//! <summary>Borrows the concrete class name for the instance lifetime. Callers must not modify it.</summary>
{attribute 'monitoring' := 'call'}
PROPERTY ClassName : REFERENCE TO STRING
GET
ClassName REF= _ClassName;
END_GET
END_PROPERTY

//! <summary>Borrows the compiler-initialized namespace. Callers must not modify it.</summary>
{attribute 'monitoring' := 'call'}
PROPERTY NamespaceName : REFERENCE TO STRING
GET
NamespaceName REF= CurrentNamespace.Name;
END_GET
END_PROPERTY

//! <summary>Reports the complete instance size in bytes, excluding separately allocated storage.</summary>
{attribute 'monitoring' := 'call'}
PROPERTY SelfSize : ULINT
GET
SelfSize := XSIZEOF(THIS^);
END_GET
END_PROPERTY

END_FUNCTION_BLOCK

// ---- Tests/Loggers/LoggerIntegrationTestGroup.TcPOU
(*
SPDX-FileCopyrightText: c 2026 Oleksandr Tiutyk <trofimich@gmail.com>
SPDX-License-Identifier: MIT
License: https://opensource.org/license/mit
*)

(*!
<summary>Groups file rotation, unfiltered file routing and native event delivery.</summary>
<description>
Owns five children in a fixed array for single-task use. Children borrows that array. The group must not be
copied.
</description>
*)

{attribute 'no_assign'}
{attribute 'no_explicit_call' := 'do not call this function block directly'}
FUNCTION_BLOCK LoggerIntegrationTestGroup EXTENDS TOF_Testing.TestGroup<5>
VAR_STAT
	{attribute 'hide'}
	_ClassName : STRING := __POUNAME();
END_VAR
VAR
	_FileRotation : TextFileLoggerRotationTest(name := "TextFileRotation", parent := THIS^);
	_EventCategories : EventLoggerCategoryTest(name := "EventCategories", parent := THIS^);
	_QueuedEvents : QueuedEventLoggerTest(name := "QueuedEvents", parent := THIS^);

	_DirectDirectory : LoggerTestDirectory(
		directoryPath := 'C:\OpenFrameworkTests\Logger_Direct',
		logFilePrefix := 'Probe'
	);
	_DirectFileLogger : TOF_Loggers.SimpleTextFileLogger(
		directoryPath := 'C:\OpenFrameworkTests\Logger_Direct',
		logFilePrefix := 'Probe',
		maxRecordsPerFile := 1,
		directoryPathType := Tc2_System.E_OpenPath.PATH_GENERIC,
		timeout := T#2S,
		amsNetId := ''
	);
	_DirectRouting : LoggerRoutingTest(
		name := "DirectFileFeedbackAndReadback",
		parent := THIS^,
		fileLogger := _DirectFileLogger,
		directory := _DirectDirectory,
		queue := 0
	);

	_QueuedDirectory : LoggerTestDirectory(
		directoryPath := 'C:\OpenFrameworkTests\Logger_Queued',
		logFilePrefix := 'Probe'
	);
	_QueuedFileLogger : TOF_Loggers.SimpleTextFileLogger(
		directoryPath := 'C:\OpenFrameworkTests\Logger_Queued',
		logFilePrefix := 'Probe',
		maxRecordsPerFile := 1,
		directoryPathType := Tc2_System.E_OpenPath.PATH_GENERIC,
		timeout := T#2S,
		amsNetId := ''
	);
	_Queue : TOF_Loggers.QueuedLogger;
	_QueuedRouting : LoggerRoutingTest(
		name := "QueuedFileFeedbackAndReadback",
		parent := THIS^,
		fileLogger := _QueuedFileLogger,
		directory := _QueuedDirectory,
		queue := _Queue
	);

	_Children : ARRAY [0.._ChildCount - 1] OF TOF_Testing.ITestElement :=
		[_FileRotation, _EventCategories, _QueuedEvents, _DirectRouting, _QueuedRouting];
END_VAR

//! <summary>Borrows the fixed child array. Callers must not modify it.</summary>
{attribute 'monitoring' := 'call'}
PROPERTY Children : REFERENCE TO ARRAY [0.._ChildCount - 1] OF TOF_Testing.ITestElement
GET
Children REF= _Children;
END_GET
END_PROPERTY

//! <summary>Borrows the concrete class name for the instance lifetime. Callers must not modify it.</summary>
{attribute 'monitoring' := 'call'}
PROPERTY ClassName : REFERENCE TO STRING
GET
ClassName REF= _ClassName;
END_GET
END_PROPERTY

//! <summary>Borrows the compiler-initialized namespace. Callers must not modify it.</summary>
{attribute 'monitoring' := 'call'}
PROPERTY NamespaceName : REFERENCE TO STRING
GET
NamespaceName REF= CurrentNamespace.Name;
END_GET
END_PROPERTY

//! <summary>Reports the complete instance size in bytes, excluding separately allocated storage.</summary>
{attribute 'monitoring' := 'call'}
PROPERTY SelfSize : ULINT
GET
SelfSize := XSIZEOF(THIS^);
END_GET
END_PROPERTY

END_FUNCTION_BLOCK

// ---- Tests/Loggers/TextFileLoggerRotationTest.TcPOU
(*
SPDX-FileCopyrightText: c 2026 Oleksandr Tiutyk <trofimich@gmail.com>
SPDX-License-Identifier: MIT
License: https://opensource.org/license/mit
*)

(*!
<summary>Checks numbered UTF-16 records and file rotation in an exclusively owned directory.</summary>
<description>
One task writes 49 records, stops the logger and reads the five generated files before removal.
A 30-second scenario deadline includes preparation and readback. Failures retain cooperative cleanup
without a forced deadline. Reset the runner only after completion.
</description>
*)

{attribute 'no_assign'}
{attribute 'no_explicit_call' := 'do not call this function block directly'}
FUNCTION_BLOCK TextFileLoggerRotationTest EXTENDS TOF_Testing.MultiCycleTest
VAR_STAT
	{attribute 'hide'}
	_ClassName : STRING := __POUNAME();
END_VAR
VAR
	_SimpleTextFileLogger : TOF_Loggers.SimpleTextFileLogger(
		directoryPath := 'C:\OpenFrameworkTests\Logger_Smoke',
		logFilePrefix := 'Log',
		maxRecordsPerFile := 10,
		directoryPathType := Tc2_System.E_OpenPath.PATH_GENERIC,
		timeout := Tc2_System.Global_Variables.DEFAULT_ADS_TIMEOUT,
		amsNetId := ''
	);
	_LogDirectory : LoggerTestDirectory(
		directoryPath := 'C:\OpenFrameworkTests\Logger_Smoke',
		logFilePrefix := 'Log'
	);
	_Phase : LOGGER_FILE_TEST_PHASE;
	_Number : ULINT;
	_Deadline : Tc2_Standard.TON;
	_Failure : TOF_Core.ERROR_MESSAGE;
	_CleanupInterrupted : BOOL;
END_VAR

(*!
<summary>Rearms the owned directory, logger and scenario clock before each run.</summary>
*)
METHOD PROTECTED BeforeTest
_Timeout := T#0S;

IF _SimpleTextFileLogger.State = TOF_Loggers.SIMPLE_TEXT_FILE_LOGGER_STATE.FAILED THEN
	RecordFailure(message := "File logger remains in terminal failure");
	RETURN;
END_IF

IF NOT _LogDirectory.Reset() THEN
	RecordFailure(message := "Cannot rearm Logger_Smoke directory after its previous run");
	RETURN;
END_IF

IF _SimpleTextFileLogger.State = TOF_Loggers.SIMPLE_TEXT_FILE_LOGGER_STATE.STOPPED THEN
	IF NOT _SimpleTextFileLogger.Start() THEN
		RecordFailure(message := "Previously stopped file logger refused Start");
		RETURN;
	END_IF
END_IF

_Phase := LOGGER_FILE_TEST_PHASE.PREPARE_DIRECTORY;
_Number := 0;
_Failure := "";
_CleanupInterrupted := FALSE;
_Deadline(IN := FALSE, PT := T#30S);
END_METHOD

(*!
<summary>Advances preparation, one numbered write, stopping or readback within the scenario deadline.</summary>
*)
METHOD PRIVATE advanceScenario
VAR
	logMessage : TOF_Core.ERROR_MESSAGE;
	expectedRecord : WSTRING(255);
END_VAR
_Deadline(IN := TRUE, PT := T#30S);

IF _Deadline.Q THEN
	_Failure := "File logger scenario exceeded 30 seconds";
	RETURN;
END_IF

CASE _Phase OF
	LOGGER_FILE_TEST_PHASE.PREPARE_DIRECTORY:
		IF FileTestRoot.FailureMessage <> TOF_Core.Strings.Empty THEN
			_Failure := TO_WSTRING(FileTestRoot.FailureMessage);
			RETURN;
		END_IF

		IF FileTestRoot.Prepared THEN
			_LogDirectory.Prepare();

			IF _LogDirectory.PreparationFailed THEN
				_Failure := TOF_Core.WideStrings.ConcatFit255(
					"Directory preparation failed: ",
					TO_WSTRING(_LogDirectory.PreparationMessage)
				);
			ELSIF _LogDirectory.Prepared THEN
				_Phase := LOGGER_FILE_TEST_PHASE.SEND_MESSAGES;
			END_IF
		END_IF

	LOGGER_FILE_TEST_PHASE.SEND_MESSAGES:
		_Number := _Number + 1;
		logMessage := TOF_Core.WideStrings.Concat255("This is log message #", TO_WSTRING(_Number));
		expectedRecord := TOF_Core.WideStrings.Concat255(
			"#",
			TO_WSTRING(_Number),
			": [INFORMATION] This is log message #",
			TO_WSTRING(_Number)
		);

		IF NOT _LogDirectory.ExpectRecord(text := expectedRecord) THEN
			_Failure := TOF_Core.WideStrings.Concat255("Cannot register expected record ", TO_WSTRING(_Number));
			RETURN;
		END_IF

		IF NOT _SimpleTextFileLogger.TryLogMessage(
			category := TOF_Core.LOG_CATEGORY.INFORMATION,
			message := logMessage,
			messageNumber := _Number
		) THEN
			_Failure := TOF_Core.WideStrings.Concat255("Logger rejected record ", TO_WSTRING(_Number));
			RETURN;
		END_IF

		_SimpleTextFileLogger.Execute();

		IF _Number = 49 THEN
			IF NOT _SimpleTextFileLogger.Stop() THEN
				_Failure := "File logger refused normal stopping";
			END_IF

			_Phase := LOGGER_FILE_TEST_PHASE.WAIT_FOR_STOP;
		END_IF

	LOGGER_FILE_TEST_PHASE.WAIT_FOR_STOP:
		_SimpleTextFileLogger.Execute();

		IF _SimpleTextFileLogger.State = TOF_Loggers.SIMPLE_TEXT_FILE_LOGGER_STATE.STOPPED THEN
			IF _SimpleTextFileLogger.Busy THEN
				_Failure := "Stopped file logger remains busy";
			ELSIF _SimpleTextFileLogger.TryLogMessage(
				category := TOF_Core.LOG_CATEGORY.INFORMATION,
				message := "after stop"
			) THEN
				_Failure := "Stopped file logger accepted a message";
			END_IF

			_Phase := LOGGER_FILE_TEST_PHASE.READBACK;
		END_IF

	LOGGER_FILE_TEST_PHASE.READBACK:
		_LogDirectory.Cleanup();

		IF _LogDirectory.CleanupComplete THEN
			IF _LogDirectory.FileCount <> 5 THEN
				_Failure := "Forty-nine records must rotate into five files";
			ELSIF _LogDirectory.LargestFileRecordCount > 10 THEN
				_Failure := "A rotated log file exceeded its ten-record limit";
			ELSIF _LogDirectory.RecordCount <> 49 THEN
				_Failure := "Readback must contain forty-nine records";
			END_IF

			_Phase := LOGGER_FILE_TEST_PHASE.COMPLETE;
		END_IF
END_CASE

IF _SimpleTextFileLogger.State = TOF_Loggers.SIMPLE_TEXT_FILE_LOGGER_STATE.FAILED AND_THEN _Failure = "" THEN
	_Failure := TOF_Core.WideStrings.ConcatFit255("File logger failed: ", _SimpleTextFileLogger.ErrorMessage);
END_IF
END_METHOD

(*!
<summary>Retains scenario failures until the logger drains and directory cleanup completes.</summary>
*)
METHOD PROTECTED ExecuteTest : TOF_Testing.TEST_CYCLE_RESULT
ExecuteTest := TOF_Testing.TEST_CYCLE_RESULT.BUSY;

IF _Phase <> LOGGER_FILE_TEST_PHASE.COMPLETE THEN
	__TRY
		advanceScenario();
	__CATCH
		_Failure := "Exception interrupted the file logger scenario";
	__ENDTRY

	IF _Failure <> "" THEN
		_Phase := LOGGER_FILE_TEST_PHASE.COMPLETE;
	END_IF

	RETURN;
END_IF

__TRY
	IF _SimpleTextFileLogger.State = TOF_Loggers.SIMPLE_TEXT_FILE_LOGGER_STATE.FAILED THEN
		IF _SimpleTextFileLogger.Busy THEN
			_SimpleTextFileLogger.Execute();
			RETURN;
		END_IF

	ELSIF _SimpleTextFileLogger.State <> TOF_Loggers.SIMPLE_TEXT_FILE_LOGGER_STATE.STOPPED THEN
		_SimpleTextFileLogger.Stop();
		_SimpleTextFileLogger.Execute();
		RETURN;
	END_IF

	_LogDirectory.Cleanup();
__CATCH
	_CleanupInterrupted := TRUE;
	RETURN;
__ENDTRY

IF NOT _LogDirectory.CleanupComplete THEN
	RETURN;
END_IF

IF _CleanupInterrupted THEN
	TOF_Core.WideStrings.AppendFit(targetString := _Failure, sourceString := " Cleanup was interrupted.");
END_IF

IF NOT _LogDirectory.CleanupSucceeded OR_ELSE _LogDirectory.CleanupMessage <> TOF_Core.Strings.Empty THEN
	TOF_Core.WideStrings.AppendFit(targetString := _Failure, sourceString := " Logger_Smoke cleanup: ");
	TOF_Core.WideStrings.AppendFit255(_Failure, TO_WSTRING(_LogDirectory.CleanupMessage));
END_IF

IF _Failure <> "" THEN
	RecordFailure(message := _Failure);
END_IF

ExecuteTest := TOF_Testing.TEST_CYCLE_RESULT.DONE;
END_METHOD

//! <summary>Borrows the concrete class name for the instance lifetime. Callers must not modify it.</summary>
{attribute 'monitoring' := 'call'}
PROPERTY ClassName : REFERENCE TO STRING
GET
ClassName REF= _ClassName;
END_GET
END_PROPERTY

//! <summary>Borrows the compiler-initialized namespace. Callers must not modify it.</summary>
{attribute 'monitoring' := 'call'}
PROPERTY NamespaceName : REFERENCE TO STRING
GET
NamespaceName REF= CurrentNamespace.Name;
END_GET
END_PROPERTY

//! <summary>Reports the complete instance size in bytes, excluding separately allocated storage.</summary>
{attribute 'monitoring' := 'call'}
PROPERTY SelfSize : ULINT
GET
SelfSize := XSIZEOF(THIS^);
END_GET
END_PROPERTY

END_FUNCTION_BLOCK

// ---- Tests/Loggers/LoggerTestDirectory.TcPOU
(*
SPDX-FileCopyrightText: © 2026 Oleksandr Tiutyk <trofimich@gmail.com>
SPDX-License-Identifier: MIT
License: https://opensource.org/license/mit
*)
(*!
<summary>Reads and removes generated log files from a newly owned test directory.</summary>
<description>
Inherits ordinary directory creation and refuses pre-existing paths. Only files matching the configured
prefix and .log suffix are registered after ownership; other entries are left untouched. The caller prevents
external directory changes and drains every logger before Cleanup. Enumeration runs to completion before
loading or deleting files. Expected short records are matched exactly once, including number and category.
Persistent native state and buffers remain alive during cleanup. Discovery is
bounded to 32 generated files; byte readback is limited to files smaller than the 8192-byte buffer.
LargestFileRecordCount reports the largest number of complete records observed in one file.
Reset rearms a fresh or successfully cleaned fixture. Errors are retained for owner inspection.
Cleanup uses nonrecursive deletion and never adopts a pre-existing directory.
</description>
*)

{attribute 'no_explicit_call' := 'do not call this function block directly'}
FUNCTION_BLOCK LoggerTestDirectory EXTENDS FileTestDirectory
VAR_STAT
	//! <summary>Concrete fixture metadata.</summary>
	_ClassName : STRING := __POUNAME();
END_VAR
VAR CONSTANT
	//! <summary>Maximum discovered artifacts; later entries remain unregistered and are not deleted.</summary>
	_MaxFiles : UINT := 32;
	//! <summary>Expected short diagnostic records retained for exact byte-readback matching.</summary>
	_MaxExpectedRecords : UINT := 50;
	//! <summary>Maximum payload code units accepted by this short-record regression fixture.</summary>
	_MaxRecordCharacters : DINT := 255;
END_VAR
VAR
	_LogFilePrefix : STRING(32);
	_LogCleanupPhase : LOGGER_DIRECTORY_CLEANUP_PHASE;
	_Enum : Tc2_Utilities.FB_EnumFindFileEntry;
	_Paths : ARRAY [0.._MaxFiles - 1] OF STRING(255);
	_FileCount : UINT;
	_FileIndex : UINT;
	_RecordCount : UDINT;
	_LargestFileRecordCount : UDINT;
	_ExpectedText : ARRAY [0.._MaxExpectedRecords - 1] OF WSTRING(255);
	_Matched : ARRAY [0.._MaxExpectedRecords - 1] OF BOOL;
	_ExpectedCount : UINT;
	_MatchedCount : UINT;
	_ReadBuffer : ARRAY [0..4095] OF WORD;
	_Load : TOF_FileSystem.LoadFile(name := "read generated log file");
	_Delete : TOF_FileSystem.DeleteFile(name := "delete owned generated log file");
	_CleanupError : STRING(255);
END_VAR

(*!
<summary>Borrows the concrete fixture type name.</summary>
<description>
Returns initialized static metadata; do not modify the referenced string.
</description>
*)
{attribute 'monitoring' := 'call'}
PROPERTY ClassName : REFERENCE TO STRING
GET
ClassName REF= _ClassName;
END_GET
END_PROPERTY

(*!
<summary>Advances discovery, byte readback and deletion after every scenario logger has drained.</summary>
<description>
Keeps incomplete native operations alive across calls. Searches only the exclusively owned directory,
registers matching regular files, then reads and deletes only those registered paths. The final inherited
cleanup attempts nonrecursive directory removal. CleanupComplete does not certify physical native release.
Readback retains the largest record count across individual files.
Matching uses exact prefix bytes and ASCII suffix/separators without computing Unicode character positions.
</description>
*)
METHOD Cleanup
VAR
	fileName : STRING(255);
	prefix : STRING(33);
	i : DINT;
	recordStart : DINT;
	fileRecordCount : UDINT;
END_VAR
IF _LogCleanupPhase = LOGGER_DIRECTORY_CLEANUP_PHASE.COMPLETE THEN
	RETURN;
END_IF

IF NOT Prepared THEN
	SUPER^.Cleanup();
	RETURN;
END_IF

__TRY

	CASE _LogCleanupPhase OF
		LOGGER_DIRECTORY_CLEANUP_PHASE.ENUMERATE_FIRST:
			_Enum(
				bExecute := FALSE,
				sNetId := '',
				sPathName := TOF_Core.Strings.Concat255(DirectoryPath, '\*'),
				ePath := Tc2_System.E_OpenPath.PATH_GENERIC,
				tTimeout := T#2S
			);
			_LogCleanupPhase := LOGGER_DIRECTORY_CLEANUP_PHASE.ENUMERATE_WAIT;
			_Enum(bExecute := TRUE, eCmd := Tc2_Utilities.E_EnumCmdType.eEnumCmd_First);

		LOGGER_DIRECTORY_CLEANUP_PHASE.ENUMERATE_WAIT:
			_Enum(bExecute := FALSE);

			IF NOT _Enum.bBusy THEN

				IF _Enum.bError THEN
					_CleanupError := TOF_Core.Strings.Concat255('Log discovery error: ', TO_STRING(_Enum.nErrId));
					_LogCleanupPhase := LOGGER_DIRECTORY_CLEANUP_PHASE.COMPLETE;
				ELSIF _Enum.bEOE THEN
					_LogCleanupPhase := LOGGER_DIRECTORY_CLEANUP_PHASE.LOAD_FILE;
				ELSE
					fileName := _Enum.stFindFile.sFileName;
					prefix := TOF_Core.Strings.Concat255(_LogFilePrefix, '_');

					IF fileName <> '.' AND_THEN fileName <> '..' THEN

						// SA0175: Exact prefix bytes and ASCII suffix/separators do not require UTF-8 character positions.
						{analysis -175}
						IF NOT _Enum.stFindFile.fileAttributes.bDirectory
							AND_THEN Tc2_Standard.LEFT(STR := fileName, SIZE := Tc2_Standard.LEN(STR := prefix)) = prefix
							AND_THEN Tc2_Standard.RIGHT(STR := fileName, SIZE := 4) = '.log'
							AND_THEN Tc2_Standard.FIND(STR1 := fileName, STR2 := '\') = 0
							AND_THEN Tc2_Standard.FIND(STR1 := fileName, STR2 := '/') = 0
							AND_THEN _FileCount < _MaxFiles
						THEN
							_Paths[_FileCount] := TOF_Core.Strings.Concat255(DirectoryPath, '\', fileName);
							_FileCount := _FileCount + 1;
						ELSE
							_CleanupError := 'Unknown or excess entry left untouched in owned log directory';
						END_IF
						{analysis +175}

					END_IF

					_LogCleanupPhase := LOGGER_DIRECTORY_CLEANUP_PHASE.ENUMERATE_NEXT;
				END_IF

			END_IF

		LOGGER_DIRECTORY_CLEANUP_PHASE.ENUMERATE_NEXT:
			_LogCleanupPhase := LOGGER_DIRECTORY_CLEANUP_PHASE.ENUMERATE_WAIT;
			_Enum(bExecute := TRUE, eCmd := Tc2_Utilities.E_EnumCmdType.eEnumCmd_Next);

		LOGGER_DIRECTORY_CLEANUP_PHASE.LOAD_FILE:

			IF _FileIndex >= _FileCount THEN
				_LogCleanupPhase := LOGGER_DIRECTORY_CLEANUP_PHASE.REMOVE_DIRECTORY;
			ELSE
				_Load.Reset();
				_Load.FilePath := _Paths[_FileIndex];
				_Load.TargetBuffer := ADR(_ReadBuffer);
				_Load.TargetBufferSize := SIZEOF(_ReadBuffer);
				_Load.Timeout := T#2S;

				IF _Load.Start() THEN
					_LogCleanupPhase := LOGGER_DIRECTORY_CLEANUP_PHASE.WAIT_FOR_LOAD;
				ELSE
					_CleanupError := 'Log readback Start refused';
					_LogCleanupPhase := LOGGER_DIRECTORY_CLEANUP_PHASE.DELETE_FILE;
				END_IF

			END_IF

		LOGGER_DIRECTORY_CLEANUP_PHASE.WAIT_FOR_LOAD:
			_Load.Execute();

			IF _Load.State.Stopped THEN

				IF NOT _Load.FinalStopReason.WorkDone THEN
					_CleanupError := 'Log byte readback failed';
				ELSIF _Load.LoadedBytesCount < 4
					OR_ELSE _Load.LoadedBytesCount >= SIZEOF(_ReadBuffer)
					OR_ELSE (_Load.LoadedBytesCount MOD 2) <> 0
					OR_ELSE _ReadBuffer[0] <> TOF_Core.WideStrings.ByteOrderMark
				THEN
					_CleanupError := 'Log bytes must contain a complete bounded UTF-16 file with BOM';
				ELSE

					recordStart := 1;
					fileRecordCount := 0;

					FOR i := 1 TO TO_DINT(_Load.LoadedBytesCount / 2) - 1 DO

						IF _ReadBuffer[i] = WORD#16#000D THEN
							_RecordCount := _RecordCount + 1;
							fileRecordCount := fileRecordCount + 1;

							IF NOT matchExpectedRecord(startIndex := recordStart, characterCount := i - recordStart) THEN
								_CleanupError := 'Readback record differs from the expected text, category or number';
							END_IF

							recordStart := i + 1;
						END_IF

					END_FOR

					_LargestFileRecordCount := MAX(_LargestFileRecordCount, fileRecordCount);

					IF _ReadBuffer[_Load.LoadedBytesCount / 2 - 1] <> WORD#16#000D THEN
						_CleanupError := 'Generated record must end with the current wide CR separator';
					END_IF

				END_IF

				_LogCleanupPhase := LOGGER_DIRECTORY_CLEANUP_PHASE.DELETE_FILE;
			END_IF

		LOGGER_DIRECTORY_CLEANUP_PHASE.DELETE_FILE:
			_Delete.Reset();
			_Delete.FilePath := _Paths[_FileIndex];
			_Delete.Timeout := T#2S;

			IF _Delete.Start() THEN
				_LogCleanupPhase := LOGGER_DIRECTORY_CLEANUP_PHASE.WAIT_FOR_DELETE;
			ELSE
				_CleanupError := 'Owned log deletion Start refused';
				_FileIndex := _FileIndex + 1;
				_LogCleanupPhase := LOGGER_DIRECTORY_CLEANUP_PHASE.LOAD_FILE;
			END_IF

		LOGGER_DIRECTORY_CLEANUP_PHASE.WAIT_FOR_DELETE:
			_Delete.Execute();

			IF _Delete.State.Stopped THEN

				IF NOT _Delete.FinalStopReason.WorkDone THEN
					_CleanupError := 'Owned log deletion failed';
				END_IF

				_FileIndex := _FileIndex + 1;
				_LogCleanupPhase := LOGGER_DIRECTORY_CLEANUP_PHASE.LOAD_FILE;
			END_IF

		LOGGER_DIRECTORY_CLEANUP_PHASE.REMOVE_DIRECTORY:
			SUPER^.Cleanup();

			IF SUPER^.CleanupComplete THEN
				_LogCleanupPhase := LOGGER_DIRECTORY_CLEANUP_PHASE.COMPLETE;
			END_IF

	END_CASE

__CATCH
	// Keep native instances and their current phase alive for the next cleanup call.
	_CleanupError := 'Exception interrupted log cleanup; keep cycling and inspect retained fixture state';
__ENDTRY
END_METHOD

(*!
<summary>Reports the owned log fixture CleanupComplete observation.</summary>
<description>
Read from the owner task. Retained results remain available after cleanup; completion does not prove
physical native resource release after an error.
</description>
*)
PROPERTY CleanupComplete : BOOL
GET
CleanupComplete := _LogCleanupPhase = LOGGER_DIRECTORY_CLEANUP_PHASE.COMPLETE OR_ELSE SUPER^.CleanupComplete;
END_GET
END_PROPERTY

(*!
<summary>Reports the owned log fixture CleanupMessage observation.</summary>
<description>
Read from the owner task. Retained results remain available after cleanup; completion does not prove
physical native resource release after an error.
</description>
*)
PROPERTY CleanupMessage : STRING(255)
GET
IF _CleanupError <> '' THEN
	CleanupMessage := _CleanupError;
ELSIF _MatchedCount <> _ExpectedCount THEN
	CleanupMessage := 'Some expected log records were not found in the generated files';
ELSE
	CleanupMessage := SUPER^.CleanupMessage;
END_IF
END_GET
END_PROPERTY

(*!
<summary>Reports the owned log fixture CleanupSucceeded observation.</summary>
<description>
Read from the owner task. Retained results remain available after cleanup; completion does not prove
physical native resource release after an error.
</description>
*)
PROPERTY CleanupSucceeded : BOOL
GET
CleanupSucceeded := SUPER^.CleanupSucceeded
	AND_THEN _CleanupError = ''
	AND_THEN _MatchedCount = _ExpectedCount;
END_GET
END_PROPERTY

(*!
<summary>Rearms a fresh or successfully cleaned logger directory for another complete readback.</summary>
<description>
Call with the logger idle. Pending or unsuccessful cleanup refuses reuse and preserves diagnostics.
Success clears prior matches and discovery counts while retaining the configured path and prefix.
</description>
*)
METHOD Reset : BOOL
VAR
	i : UINT;
END_VAR
IF CleanupComplete AND_THEN NOT CleanupSucceeded THEN
	RETURN;
END_IF

IF NOT SUPER^.Reset() THEN
	RETURN;
END_IF

FOR i := 0 TO _MaxExpectedRecords - 1 DO
	_Matched[i] := FALSE;
END_FOR

_FileCount := 0;
_FileIndex := 0;
_RecordCount := 0;
_LargestFileRecordCount := 0;
_ExpectedCount := 0;
_MatchedCount := 0;
_CleanupError := TOF_Core.Strings.Empty;
_LogCleanupPhase := LOGGER_DIRECTORY_CLEANUP_PHASE.ENUMERATE_FIRST;
Reset := TRUE;
END_METHOD

(*!
<summary>Registers one independently specified short record before the logger may write it.</summary>
<description>
Call only after directory ownership is established and before Cleanup. Copies up to 255 code units; returns
FALSE before preparation or when fifty expected records are already stored. Readback matches every record
exactly once, independently of native enumeration order. Inputs in these scenarios contain no embedded CR.
</description>
*)
METHOD ExpectRecord : BOOL
VAR_INPUT
	text : WSTRING(255);
END_VAR
IF NOT Prepared OR_ELSE _ExpectedCount >= _MaxExpectedRecords THEN
	RETURN;
END_IF

_ExpectedText[_ExpectedCount] := text;
_ExpectedCount := _ExpectedCount + 1;
ExpectRecord := TRUE;
END_METHOD

(*!
<summary>Copies the permitted artifact prefix without performing I/O.</summary>
<description>
The base receives directoryPath implicitly. Both additional arguments are mandatory at initialization;
logFilePrefix must equal the logger prefix used exclusively inside the owned scenario directory.
</description>
*)
METHOD FB_init : BOOL
VAR_INPUT
	bInitRetains : BOOL; // TRUE: the retain variables are initialized (reset warm / reset cold)
	bInCopyCode : BOOL; // TRUE: the instance will be copied to the copy code afterward (online change)
	directoryPath : STRING(255);
	logFilePrefix : STRING(32);
END_VAR
IF NOT bInCopyCode THEN
	_LogFilePrefix := logFilePrefix;
END_IF
END_METHOD

(*!
<summary>Reports the owned log fixture FileCount observation.</summary>
<description>
Read from the owner task. Retained results remain available after cleanup; completion does not prove
physical native resource release after an error.
</description>
*)
PROPERTY FileCount : UINT
GET
FileCount := _FileCount;
END_GET
END_PROPERTY

(*!
<summary>Matches one complete short UTF-16 record to a not-yet-consumed expected value.</summary>
<description>
Called only with a validated byte buffer and the range between two observed wide CR separators. Copies
no more than 255 code units into local passive storage and writes its terminator explicitly. Enumeration
order does not affect matching; each expected value can be consumed at most once.
</description>
*)
METHOD PRIVATE matchExpectedRecord : BOOL
VAR_INPUT
	startIndex : DINT;
	characterCount : DINT;
END_VAR
VAR
	record : WSTRING(255);
	recordWords : POINTER TO WORD;
	j : DINT;
END_VAR
IF characterCount > _MaxRecordCharacters THEN
	RETURN;
END_IF

Tc2_System.MEMCPY(
	destAddr := ADR(record),
	srcAddr := ADR(_ReadBuffer[startIndex]),
	n := TO_UDINT(characterCount * TOF_Core.WideStrings.CharSize)
);
recordWords := ADR(record);
// Terminate the copied UTF-16 record independently of previous buffer contents.
recordWords[characterCount] := 0;

FOR j := 0 TO TO_DINT(_ExpectedCount) - 1 DO

	IF NOT _Matched[j] AND_THEN _ExpectedText[j] = record THEN
		_Matched[j] := TRUE;
		_MatchedCount := _MatchedCount + 1;
		matchExpectedRecord := TRUE;
		RETURN;
	END_IF

END_FOR
END_METHOD

(*!
<summary>Borrows the test namespace.</summary>
<description>
Returns compiler-initialized library storage without ownership transfer.
</description>
*)
{attribute 'monitoring' := 'call'}
PROPERTY NamespaceName : REFERENCE TO STRING
GET
NamespaceName REF= CurrentNamespace.Name;
END_GET
END_PROPERTY

(*!
<summary>Reports the maximum count of wide-CR records read from a single generated file.</summary>
<description>Accumulates during cleanup and returns to zero on successful Reset.</description>
*)
PROPERTY LargestFileRecordCount : UDINT
GET
LargestFileRecordCount := _LargestFileRecordCount;
END_GET
END_PROPERTY

(*!
<summary>Reports the owned log fixture RecordCount observation.</summary>
<description>
Read from the owner task. Retained results remain available after cleanup; completion does not prove
physical native resource release after an error.
</description>
*)
PROPERTY RecordCount : UDINT
GET
RecordCount := _RecordCount;
END_GET
END_PROPERTY

(*!
<summary>Reports the concrete fixture size in bytes.</summary>
*)
{attribute 'monitoring' := 'call'}
PROPERTY SelfSize : ULINT
GET
SelfSize := XSIZEOF(THIS^);
END_GET
END_PROPERTY

END_FUNCTION_BLOCK

// ---- Tests/Loggers/EventLoggerCategoryTest.TcPOU
(*
SPDX-FileCopyrightText: c 2026 Oleksandr Tiutyk <trofimich@gmail.com>
SPDX-License-Identifier: MIT
License: https://opensource.org/license/mit
*)

(*!
<summary>Exercises all five native event categories.</summary>
<description>
Each run submits five numbered messages from the runner task and checks each admission result.
</description>
*)

{attribute 'no_assign'}
{attribute 'no_explicit_call' := 'do not call this function block directly'}
FUNCTION_BLOCK EventLoggerCategoryTest EXTENDS TOF_Testing.SingleCycleTest
VAR_STAT
	{attribute 'hide'}
	_ClassName : STRING := __POUNAME();
END_VAR
VAR
	_EventLogger : TOF_Loggers.EventLogger(
		debugEventType := TC_EVENTS.OpenFrameworkLoggerEventClass.DebugEvent,
		informationEventType := TC_EVENTS.OpenFrameworkLoggerEventClass.InformationEvent,
		warningEventType := TC_EVENTS.OpenFrameworkLoggerEventClass.WarningEvent,
		errorEventType := TC_EVENTS.OpenFrameworkLoggerEventClass.ErrorEvent,
		criticalErrorEventType := TC_EVENTS.OpenFrameworkLoggerEventClass.CriticalErrorEvent
	);
END_VAR

(*!
<summary>Sends a numbered message for each configured event type and checks the native result.</summary>
*)
METHOD PROTECTED ExecuteTest
VAR
	number : ULINT;
END_VAR
number := 1;
Assert.ThatBool(
	actual := _EventLogger.TryLogMessage(
		category := TOF_Core.LOG_CATEGORY.DEBUG,
		message := "LoggerTest DEBUG",
		messageNumber := number
	),
	message := "EventLogger refused DEBUG"
).IsTrue();

number := 2;
Assert.ThatBool(
	actual := _EventLogger.TryLogMessage(
		category := TOF_Core.LOG_CATEGORY.INFORMATION,
		message := "LoggerTest INFORMATION",
		messageNumber := number
	),
	message := "EventLogger refused INFORMATION"
).IsTrue();

number := 3;
Assert.ThatBool(
	actual := _EventLogger.TryLogMessage(
		category := TOF_Core.LOG_CATEGORY.WARNING,
		message := "LoggerTest WARNING",
		messageNumber := number
	),
	message := "EventLogger refused WARNING"
).IsTrue();

number := 4;
Assert.ThatBool(
	actual := _EventLogger.TryLogMessage(
		category := TOF_Core.LOG_CATEGORY.ERROR,
		message := "LoggerTest ERROR",
		messageNumber := number
	),
	message := "EventLogger refused ERROR"
).IsTrue();

number := 5;
Assert.ThatBool(
	actual := _EventLogger.TryLogMessage(
		category := TOF_Core.LOG_CATEGORY.CRITICAL_ERROR,
		message := "LoggerTest CRITICAL_ERROR",
		messageNumber := number
	),
	message := "EventLogger refused CRITICAL_ERROR"
).IsTrue();
END_METHOD

//! <summary>Borrows the concrete class name for the instance lifetime. Callers must not modify it.</summary>
{attribute 'monitoring' := 'call'}
PROPERTY ClassName : REFERENCE TO STRING
GET
ClassName REF= _ClassName;
END_GET
END_PROPERTY

//! <summary>Borrows the compiler-initialized namespace. Callers must not modify it.</summary>
{attribute 'monitoring' := 'call'}
PROPERTY NamespaceName : REFERENCE TO STRING
GET
NamespaceName REF= CurrentNamespace.Name;
END_GET
END_PROPERTY

//! <summary>Reports the complete instance size in bytes, excluding separately allocated storage.</summary>
{attribute 'monitoring' := 'call'}
PROPERTY SelfSize : ULINT
GET
SelfSize := XSIZEOF(THIS^);
END_GET
END_PROPERTY

END_FUNCTION_BLOCK

// ---- Tests/Loggers/QueuedEventLoggerTest.TcPOU
(*
SPDX-FileCopyrightText: c 2026 Oleksandr Tiutyk <trofimich@gmail.com>
SPDX-License-Identifier: MIT
License: https://opensource.org/license/mit
*)

(*!
<summary>Checks queued delivery to the native EventLogger.</summary>
<description>
The runner task owns the configured queue and backend for every run.
</description>
*)

{attribute 'no_assign'}
{attribute 'no_explicit_call' := 'do not call this function block directly'}
FUNCTION_BLOCK QueuedEventLoggerTest EXTENDS TOF_Testing.SingleCycleTest
VAR_STAT
	{attribute 'hide'}
	_ClassName : STRING := __POUNAME();
END_VAR
VAR
	_EventLogger : TOF_Loggers.EventLogger(
		debugEventType := TC_EVENTS.OpenFrameworkLoggerEventClass.DebugEvent,
		informationEventType := TC_EVENTS.OpenFrameworkLoggerEventClass.InformationEvent,
		warningEventType := TC_EVENTS.OpenFrameworkLoggerEventClass.WarningEvent,
		errorEventType := TC_EVENTS.OpenFrameworkLoggerEventClass.ErrorEvent,
		criticalErrorEventType := TC_EVENTS.OpenFrameworkLoggerEventClass.CriticalErrorEvent
	);
	_Queue : TOF_Loggers.QueuedLogger;
	_Configured : BOOL;
END_VAR

(*!
<summary>Submits two messages and a copied error to the queue and checks delivery to EventLogger.</summary>
*)
METHOD PROTECTED ExecuteTest
VAR
	number : ULINT := 1;
	error : TOF_Core.ERROR;
	failuresBefore : ULINT;
END_VAR
failuresBefore := _Queue.FailedDeliveryCount;

IF NOT _Configured THEN
	Assert.ThatULInt(actual := failuresBefore, message := "A fresh queue must have zero delivery failures").ToBe(
		expected := 0
	);
	_Configured := _Queue.Configure(backend := _EventLogger);
END_IF

IF NOT _Configured THEN
	RecordFailure(message := "Queue refused the EventLogger backend");
	RETURN;
END_IF

Assert.ThatDInt(actual := _Queue.PendingMessageCount, message := "Queue must start empty").ToBe(expected := 0);
Assert.ThatBool(
	actual := _Queue.TryLogMessage(category := TOF_Core.LOG_CATEGORY.DEBUG, message := "Queued debug message"),
	message := "Queue refused the unnumbered debug message"
).IsTrue();
Assert.ThatDInt(actual := _Queue.PendingMessageCount, message := "Debug message must be pending").ToBe(expected := 1);
Assert.ThatBool(
	actual := _Queue.TryLogMessage(
		category := TOF_Core.LOG_CATEGORY.INFORMATION,
		message := "Queued information message",
		messageNumber := number
	),
	message := "Queue refused the numbered information message"
).IsTrue();
Assert.ThatDInt(actual := _Queue.PendingMessageCount, message := "Both messages must be pending").ToBe(expected := 2);
error.SetMessage(message := "Queued error");
error.SetSeverity(severity := TOF_Core.ERROR_SEVERITY.ERROR);
Assert.ThatBool(
	actual := _Queue.TryLogError(error := error, messageNumber := number),
	message := "Queue refused the error record"
).IsTrue();
Assert.ThatDInt(actual := _Queue.PendingMessageCount, message := "Three records must be pending").ToBe(expected := 3);
_Queue.Execute();
Assert.ThatDInt(actual := _Queue.PendingMessageCount, message := "Native batch must drain").ToBe(expected := 0);
Assert.ThatULInt(actual := _Queue.FailedDeliveryCount, message := "EventLogger must accept every queued record").ToBe(
	expected := failuresBefore
);
END_METHOD

//! <summary>Borrows the concrete class name for the instance lifetime. Callers must not modify it.</summary>
{attribute 'monitoring' := 'call'}
PROPERTY ClassName : REFERENCE TO STRING
GET
ClassName REF= _ClassName;
END_GET
END_PROPERTY

//! <summary>Borrows the compiler-initialized namespace. Callers must not modify it.</summary>
{attribute 'monitoring' := 'call'}
PROPERTY NamespaceName : REFERENCE TO STRING
GET
NamespaceName REF= CurrentNamespace.Name;
END_GET
END_PROPERTY

//! <summary>Reports the complete instance size in bytes, excluding separately allocated storage.</summary>
{attribute 'monitoring' := 'call'}
PROPERTY SelfSize : ULINT
GET
SelfSize := XSIZEOF(THIS^);
END_GET
END_PROPERTY

END_FUNCTION_BLOCK

// ---- Tests/Loggers/LoggerRoutingTest.TcPOU
(*
SPDX-FileCopyrightText: c 2026 Oleksandr Tiutyk <trofimich@gmail.com>
SPDX-License-Identifier: MIT
License: https://opensource.org/license/mit
*)

(*!
<summary>Checks that file logger service produces only the two external records when routed through LogManager.</summary>
<description>
Each instance exclusively drives its parent-owned directory and file logger, optionally through a dedicated queue.
Requires single-task use and no concurrent logging or filter changes during the temporary unfiltered service calls.
Observes eight consecutive idle calls before Stop. The 30-second deadline includes preparation and readback.
Failures retain cooperative cleanup. Reset only after completion. Do not copy an instance or its borrowed fixtures.
</description>
*)

{attribute 'no_explicit_call' := 'do not call this function block directly'}
FUNCTION_BLOCK LoggerRoutingTest EXTENDS TOF_Testing.MultiCycleTest
VAR_STAT
	{attribute 'hide'}
	_ClassName : STRING := __POUNAME();
END_VAR
VAR
	_FileLogger : REFERENCE TO TOF_Loggers.SimpleTextFileLogger;
	_Directory : REFERENCE TO LoggerTestDirectory;
	_Queue : REFERENCE TO TOF_Loggers.QueuedLogger;
	_Route : TOF_Core.ILogger;
	_QueueConfigured : BOOL;
	_FailuresBefore : ULINT;
	_Phase : LOGGER_FILE_TEST_PHASE;
	_IdleCycles : UINT;
	_Deadline : Tc2_Standard.TON;
	_Failure : TOF_Core.ERROR_MESSAGE;
	_CleanupInterrupted : BOOL;
END_VAR

(*!
<summary>Borrows fixtures dedicated to this case. Performs no I/O.</summary>
<param name="name">Case name in reports.</param>
<param name="parent">Owning group.</param>
<param name="fileLogger">File backend configured for one record per file.</param>
<param name="directory">Exclusive fixture with the same directory and prefix as the backend.</param>
<param name="queue">Dedicated queue, or a null reference for direct service.</param>
*)
METHOD FB_init : BOOL
VAR_INPUT
	bInitRetains: BOOL; // TRUE: the retain variables are initialized (reset warm / reset cold)
	bInCopyCode: BOOL; // TRUE: the instance will be copied to the copy code afterward (online change)
	name : WSTRING;
	parent : TOF_Testing.ITestElement;
	fileLogger : REFERENCE TO TOF_Loggers.SimpleTextFileLogger;
	directory : REFERENCE TO LoggerTestDirectory;
	queue : REFERENCE TO TOF_Loggers.QueuedLogger;
END_VAR
IF NOT bInCopyCode THEN
	_FileLogger REF= fileLogger;
	_Directory REF= directory;
	_Queue REF= queue;
END_IF

FB_init := TRUE;
END_METHOD

(*!
<summary>Services the current task logger with the manager filter temporarily disabled.</summary>
<description>
Saves and restores this task's logger and the shared filter within this synchronous call. Tests require no
concurrent logging while changing the shared filter. Restoring a standard logger view preserves its behavior
when previously unset.
The independent embedded diagnostic channel must not reenter this LogManager call.
An exception during service is reported after the route is restored and cleanup completes.
</description>
<param name="logger">Temporary service destination.</param>
*)
METHOD PRIVATE executeWithRouting
VAR_INPUT
	logger : TOF_Core.ILogger;
END_VAR
VAR
	savedLogger : TOF_Core.ILogger;
	savedFilter : TOF_Core.ILogFilter;
END_VAR
savedLogger := TOF_Core.LogManager.CurrentTaskLogger;
savedFilter := TOF_Core.LogManager.Filter;

__TRY
	TOF_Core.LogManager.CurrentTaskLogger := logger;
	TOF_Core.LogManager.Filter := 0;
	TOF_Core.LogManager.ExecuteCurrentTaskLogger();
__CATCH
	_Failure := "Current-task logger service raised an exception";
__ENDTRY

TOF_Core.LogManager.Filter := savedFilter;
TOF_Core.LogManager.CurrentTaskLogger := savedLogger;
END_METHOD

(*!
<summary>Rearms the owned directory, logger and scenario clock before each run.</summary>
*)
METHOD PROTECTED BeforeTest
_Timeout := T#0S;

IF NOT __ISVALIDREF(_Directory) OR_ELSE NOT __ISVALIDREF(_FileLogger) THEN
	RecordFailure(message := "Routed file test requires both directory and file logger");
	RETURN;
END_IF

_Route := _FileLogger;

IF __ISVALIDREF(_Queue) THEN
	IF NOT _QueueConfigured THEN
		_QueueConfigured := _Queue.Configure(backend := _FileLogger);
	END_IF

	IF NOT _QueueConfigured OR_ELSE _Queue.PendingMessageCount <> 0 THEN
		RecordFailure(message := "Queue must be configured and empty before the scenario");
		RETURN;
	END_IF

	_Route := _Queue;
	_FailuresBefore := _Queue.FailedDeliveryCount;
END_IF

IF _FileLogger.State = TOF_Loggers.SIMPLE_TEXT_FILE_LOGGER_STATE.FAILED THEN
	RecordFailure(message := "File logger remains in terminal failure");
	RETURN;
END_IF

IF NOT _Directory.Reset() THEN
	RecordFailure(message := "Cannot rearm routed logger directory after its previous run");
	RETURN;
END_IF

IF _FileLogger.State = TOF_Loggers.SIMPLE_TEXT_FILE_LOGGER_STATE.STOPPED THEN
	IF NOT _FileLogger.Start() THEN
		RecordFailure(message := "Previously stopped file logger refused Start");
		RETURN;
	END_IF
END_IF

_Phase := LOGGER_FILE_TEST_PHASE.PREPARE_DIRECTORY;
_IdleCycles := 0;
_Failure := "";
_CleanupInterrupted := FALSE;
_Deadline(IN := FALSE, PT := T#30S);
END_METHOD

(*!
<summary>Advances route admission, idle observation, stopping and file readback within the deadline.</summary>
*)
METHOD PRIVATE advanceScenario
VAR
	number : ULINT;
END_VAR
_Deadline(IN := TRUE, PT := T#30S);

IF _Deadline.Q THEN
	_Failure := "File logger scenario exceeded 30 seconds";
	RETURN;
END_IF

CASE _Phase OF
	LOGGER_FILE_TEST_PHASE.PREPARE_DIRECTORY:
		IF FileTestRoot.FailureMessage <> TOF_Core.Strings.Empty THEN
			_Failure := TO_WSTRING(FileTestRoot.FailureMessage);
			RETURN;
		END_IF

		IF FileTestRoot.Prepared THEN
			_Directory.Prepare();

			IF _Directory.PreparationFailed THEN
				_Failure := TOF_Core.WideStrings.ConcatFit255(
					"Directory preparation failed: ",
					TO_WSTRING(_Directory.PreparationMessage)
				);
			ELSIF _Directory.Prepared THEN
				_Phase := LOGGER_FILE_TEST_PHASE.SEND_MESSAGES;
			END_IF
		END_IF

	LOGGER_FILE_TEST_PHASE.SEND_MESSAGES:
		IF NOT _Directory.ExpectRecord(text := "#41: [INFORMATION] first routed record")
			OR_ELSE NOT _Directory.ExpectRecord(text := "#42: [INFORMATION] second routed record")
		THEN
			_Failure := "Cannot register the two expected records";
			RETURN;
		END_IF

		number := 41;

		IF NOT _Route.TryLogMessage(
			category := TOF_Core.LOG_CATEGORY.INFORMATION,
			message := "first routed record",
			messageNumber := number
		) THEN
			_Failure := "Route rejected record 41";
			RETURN;
		END_IF

		number := 42;

		IF NOT _Route.TryLogMessage(
			category := TOF_Core.LOG_CATEGORY.INFORMATION,
			message := "second routed record",
			messageNumber := number
		) THEN
			_Failure := "Route rejected record 42";
			RETURN;
		END_IF

		IF __ISVALIDREF(_Queue) AND_THEN _Queue.PendingMessageCount <> 2 THEN
			_Failure := "Both queued records must be pending before the first service call";
			RETURN;
		END_IF

		_Phase := LOGGER_FILE_TEST_PHASE.OBSERVE_IDLE;

	LOGGER_FILE_TEST_PHASE.OBSERVE_IDLE:
		executeWithRouting(logger := _Route);

		IF _FileLogger.Busy OR_ELSE (__ISVALIDREF(_Queue) AND_THEN _Queue.PendingMessageCount <> 0) THEN
			_IdleCycles := 0;
		ELSE
			_IdleCycles := _IdleCycles + 1;

			IF _IdleCycles = 8 THEN
				IF NOT _FileLogger.Stop() THEN
					_Failure := "Idle routed file logger refused Stop";
				END_IF

				_Phase := LOGGER_FILE_TEST_PHASE.WAIT_FOR_STOP;
			END_IF
		END_IF

	LOGGER_FILE_TEST_PHASE.WAIT_FOR_STOP:
		executeWithRouting(logger := _Route);

		IF _FileLogger.State = TOF_Loggers.SIMPLE_TEXT_FILE_LOGGER_STATE.STOPPED THEN
			IF _FileLogger.Busy THEN
				_Failure := "Stopped file logger remains busy";
			ELSIF __ISVALIDREF(_Queue)
				AND_THEN (_Queue.PendingMessageCount <> 0 OR_ELSE _Queue.FailedDeliveryCount <> _FailuresBefore)
			THEN
				_Failure := "Queued route retained or failed a delivery";
			END_IF

			_Phase := LOGGER_FILE_TEST_PHASE.READBACK;
		END_IF

	LOGGER_FILE_TEST_PHASE.READBACK:
		_Directory.Cleanup();

		IF _Directory.CleanupComplete THEN
			IF _Directory.FileCount <> 2 THEN
				_Failure := "Two external records must create exactly two files";
			ELSIF _Directory.LargestFileRecordCount <> 1 THEN
				_Failure := "Each file must contain one routed record";
			ELSIF _Directory.RecordCount <> 2 THEN
				_Failure := "Readback must contain exactly two external records";
			END_IF

			_Phase := LOGGER_FILE_TEST_PHASE.COMPLETE;
		END_IF
END_CASE

IF _FileLogger.State = TOF_Loggers.SIMPLE_TEXT_FILE_LOGGER_STATE.FAILED AND_THEN _Failure = "" THEN
	_Failure := TOF_Core.WideStrings.ConcatFit255("File logger failed: ", _FileLogger.ErrorMessage);
END_IF
END_METHOD

(*!
<summary>Retains scenario failures until the logger drains and directory cleanup completes.</summary>
*)
METHOD PROTECTED ExecuteTest : TOF_Testing.TEST_CYCLE_RESULT
ExecuteTest := TOF_Testing.TEST_CYCLE_RESULT.BUSY;

IF _Phase <> LOGGER_FILE_TEST_PHASE.COMPLETE THEN
	__TRY
		advanceScenario();
	__CATCH
		_Failure := "Exception interrupted the file logger scenario";
	__ENDTRY

	IF _Failure <> "" THEN
		_Phase := LOGGER_FILE_TEST_PHASE.COMPLETE;
	END_IF

	RETURN;
END_IF

__TRY
	IF __ISVALIDREF(_Queue) AND_THEN _Queue.PendingMessageCount <> 0 THEN
		_Queue.Execute();
		RETURN;
	END_IF

	IF _FileLogger.State = TOF_Loggers.SIMPLE_TEXT_FILE_LOGGER_STATE.FAILED THEN
		IF _FileLogger.Busy THEN
			_FileLogger.Execute();
			RETURN;
		END_IF

	ELSIF _FileLogger.State <> TOF_Loggers.SIMPLE_TEXT_FILE_LOGGER_STATE.STOPPED THEN
		_FileLogger.Stop();
		_FileLogger.Execute();
		RETURN;
	END_IF

	_Directory.Cleanup();
__CATCH
	_CleanupInterrupted := TRUE;
	RETURN;
__ENDTRY

IF NOT _Directory.CleanupComplete THEN
	RETURN;
END_IF

IF _CleanupInterrupted THEN
	TOF_Core.WideStrings.AppendFit(targetString := _Failure, sourceString := " Cleanup was interrupted.");
END_IF

IF NOT _Directory.CleanupSucceeded OR_ELSE _Directory.CleanupMessage <> TOF_Core.Strings.Empty THEN
	TOF_Core.WideStrings.AppendFit(targetString := _Failure, sourceString := " routed logger cleanup: ");
	TOF_Core.WideStrings.AppendFit255(_Failure, TO_WSTRING(_Directory.CleanupMessage));
END_IF

IF _Failure <> "" THEN
	RecordFailure(message := _Failure);
END_IF

ExecuteTest := TOF_Testing.TEST_CYCLE_RESULT.DONE;
END_METHOD

//! <summary>Borrows the concrete class name for the instance lifetime. Callers must not modify it.</summary>
{attribute 'monitoring' := 'call'}
PROPERTY ClassName : REFERENCE TO STRING
GET
ClassName REF= _ClassName;
END_GET
END_PROPERTY

//! <summary>Borrows the compiler-initialized namespace. Callers must not modify it.</summary>
{attribute 'monitoring' := 'call'}
PROPERTY NamespaceName : REFERENCE TO STRING
GET
NamespaceName REF= CurrentNamespace.Name;
END_GET
END_PROPERTY

//! <summary>Reports the complete instance size in bytes, excluding separately allocated storage.</summary>
{attribute 'monitoring' := 'call'}
PROPERTY SelfSize : ULINT
GET
SelfSize := XSIZEOF(THIS^);
END_GET
END_PROPERTY

END_FUNCTION_BLOCK

// ---- Tests/Tasks/TaskLifecycleViewsTestGroup.TcPOU
(*
SPDX-FileCopyrightText: © 2026 Oleksandr Tiutyk <trofimich@gmail.com>
SPDX-License-Identifier: MIT
License: https://opensource.org/license/mit
*)

(*!
<summary>Groups the task lifecycle view and naming cases.</summary>
<description>
Owns the child cases and their fixed registration array. Use from one task. The group must not be copied.
</description>
*)

{attribute 'no_assign'}
{attribute 'no_explicit_call' := 'do not call this function block directly'}
FUNCTION_BLOCK TaskLifecycleViewsTestGroup EXTENDS TOF_Testing.TestGroup<8>
VAR_STAT
	{attribute 'hide'}
	_ClassName : STRING := __POUNAME();
END_VAR
VAR
	_UnboundTaskState : UnboundTaskStateTest(
		name := "UnboundTaskStateDoesNotFault",
		parent := THIS^
	);
	_TaskStateView : BoundTaskStateTest(
		name := "TaskStateTracksLiveVariables",
		parent := THIS^
	);
	_UnboundTaskRunningSubstate : UnboundTaskRunningSubstateTest(
		name := "UnboundTaskRunningSubstateDoesNotFault",
		parent := THIS^
	);
	_TaskRunningSubstateView : BoundTaskRunningSubstateTest(
		name := "TaskRunningSubstateTracksLiveVariables",
		parent := THIS^
	);
	_UnboundTaskStopReason : UnboundTaskStopReasonTest(
		name := "UnboundTaskStopReasonDoesNotFault",
		parent := THIS^
	);
	_TaskStopReasonView : BoundTaskStopReasonTest(
		name := "TaskStopReasonTracksLiveVariables",
		parent := THIS^
	);
	_Reinitialization : TaskReinitViewsTest(
		name := "TaskFBReinitPreservesLiveViews",
		parent := THIS^
	);
	_NamePreservedByReset : TaskNamePreservedByResetTest(
		name := "TaskNamePreservedByReset",
		parent := THIS^
	);

	_Children : ARRAY [0.._ChildCount - 1] OF TOF_Testing.ITestElement :=
	[
		_UnboundTaskState,
		_TaskStateView,
		_UnboundTaskRunningSubstate,
		_TaskRunningSubstateView,
		_UnboundTaskStopReason,
		_TaskStopReasonView,
		_Reinitialization,
		_NamePreservedByReset
	];
END_VAR

//! <summary>Borrows the fixed child array. Callers must not modify it.</summary>
{attribute 'monitoring' := 'call'}
PROPERTY Children : REFERENCE TO ARRAY [0.._ChildCount - 1] OF TOF_Testing.ITestElement
GET
Children REF= _Children;
END_GET
END_PROPERTY

//! <summary>Borrows the concrete class name. Callers must not modify the returned storage.</summary>
{attribute 'monitoring' := 'call'}
PROPERTY ClassName : REFERENCE TO STRING
GET
ClassName REF= _ClassName;
END_GET
END_PROPERTY

//! <summary>Borrows the compiler-initialized namespace name. Callers must not modify the returned storage.</summary>
{attribute 'monitoring' := 'call'}
PROPERTY NamespaceName : REFERENCE TO STRING
GET
NamespaceName REF= CurrentNamespace.Name;
END_GET
END_PROPERTY

//! <summary>Reports the complete concrete instance size in bytes.</summary>
{attribute 'monitoring' := 'call'}
PROPERTY SelfSize : ULINT
GET
SelfSize := XSIZEOF(THIS^);
END_GET
END_PROPERTY

END_FUNCTION_BLOCK

// ---- Tests/Tasks/UnboundTaskStateTest.TcPOU
(*
SPDX-FileCopyrightText: © 2026 Oleksandr Tiutyk <trofimich@gmail.com>
SPDX-License-Identifier: MIT
License: https://opensource.org/license/mit
*)

(*!
<summary>Checks safe defaults for an unbound TaskState view.</summary>
<description>
Uses unbound local references and checks every observable property without dereferencing a missing target.
</description>
*)

{attribute 'no_explicit_call' := 'do not call this function block directly'}
FUNCTION_BLOCK UnboundTaskStateTest EXTENDS TOF_Testing.SingleCycleTest
VAR_STAT
	{attribute 'hide'}
	_ClassName : STRING := __POUNAME();
END_VAR

//! <summary>Reads all flags and verifies the default value for an unbound view.</summary>
METHOD PROTECTED ExecuteTest
VAR
	backingValue : REFERENCE TO TOF_Tasks.TASK_STATE;
	stateChanged : REFERENCE TO BOOL;
	view : TOF_Tasks.TaskState(taskState := backingValue, taskStateChanged := stateChanged);
END_VAR
Assert.ThatBool(actual := view.Ready, message := "Unbound TaskState.Ready must be false").IsFalse();
Assert.ThatBool(actual := view.Running, message := "Unbound TaskState.Running must be false").IsFalse();
Assert.ThatBool(actual := view.Stopped, message := "Unbound TaskState.Stopped must be false").IsFalse();
Assert.ThatBool(actual := view.StateChanged, message := "Unbound TaskState.StateChanged must be false").IsFalse();
Assert.ThatBool(
	actual := view.Value = TOF_Tasks.TASK_STATE.READY,
	message := "Unbound Value must default to READY"
).IsTrue();
END_METHOD

//! <summary>Borrows the concrete class name. Callers must not modify the returned storage.</summary>
{attribute 'monitoring' := 'call'}
PROPERTY ClassName : REFERENCE TO STRING
GET
ClassName REF= _ClassName;
END_GET
END_PROPERTY

//! <summary>Borrows the compiler-initialized namespace name. Callers must not modify the returned storage.</summary>
{attribute 'monitoring' := 'call'}
PROPERTY NamespaceName : REFERENCE TO STRING
GET
NamespaceName REF= CurrentNamespace.Name;
END_GET
END_PROPERTY

//! <summary>Reports the complete concrete instance size in bytes.</summary>
{attribute 'monitoring' := 'call'}
PROPERTY SelfSize : ULINT
GET
SelfSize := XSIZEOF(THIS^);
END_GET
END_PROPERTY

END_FUNCTION_BLOCK

// ---- Tests/Tasks/BoundTaskStateTest.TcPOU
(*
SPDX-FileCopyrightText: © 2026 Oleksandr Tiutyk <trofimich@gmail.com>
SPDX-License-Identifier: MIT
License: https://opensource.org/license/mit
*)

(*!
<summary>Checks that a bound TaskState view observes changes to its backing data.</summary>
<description>
Exercises all defined values through the same view in one call. The backing data and view are local to the call.
</description>
*)

{attribute 'no_explicit_call' := 'do not call this function block directly'}
FUNCTION_BLOCK BoundTaskStateTest EXTENDS TOF_Testing.SingleCycleTest
VAR_STAT
	{attribute 'hide'}
	_ClassName : STRING := __POUNAME();
END_VAR

//! <summary>Sets each backing value and checks the corresponding value and flags.</summary>
METHOD PROTECTED ExecuteTest
VAR
	backingValue : TOF_Tasks.TASK_STATE;
	stateChanged : BOOL;
	view : TOF_Tasks.TaskState(taskState := backingValue, taskStateChanged := stateChanged);
END_VAR
backingValue := TOF_Tasks.TASK_STATE.READY;
stateChanged := FALSE;
Assert.ThatBool(actual := view.Value = TOF_Tasks.TASK_STATE.READY, message := "Value must track READY").IsTrue();
Assert.ThatBool(actual := view.Ready, message := "Ready must be true for READY").IsTrue();
Assert.ThatBool(actual := view.Running, message := "Running must be false for READY").IsFalse();
Assert.ThatBool(actual := view.Stopped, message := "Stopped must be false for READY").IsFalse();
Assert.ThatBool(actual := view.StateChanged, message := "StateChanged must track its backing flag in READY").IsFalse();

backingValue := TOF_Tasks.TASK_STATE.RUNNING;
stateChanged := TRUE;
Assert.ThatBool(actual := view.Value = TOF_Tasks.TASK_STATE.RUNNING, message := "Value must track RUNNING").IsTrue();
Assert.ThatBool(actual := view.Running, message := "Running must be true for RUNNING").IsTrue();
Assert.ThatBool(actual := view.Ready, message := "Ready must be false for RUNNING").IsFalse();
Assert.ThatBool(actual := view.Stopped, message := "Stopped must be false for RUNNING").IsFalse();
Assert.ThatBool(actual := view.StateChanged, message := "StateChanged must track its backing flag in RUNNING").IsTrue();

stateChanged := FALSE;
Assert.ThatBool(
	actual := view.StateChanged,
	message := "StateChanged must clear while the lifecycle state stays RUNNING"
).IsFalse();

backingValue := TOF_Tasks.TASK_STATE.STOPPED;
stateChanged := FALSE;
Assert.ThatBool(actual := view.Value = TOF_Tasks.TASK_STATE.STOPPED, message := "Value must track STOPPED").IsTrue();
Assert.ThatBool(actual := view.Stopped, message := "Stopped must be true for STOPPED").IsTrue();
Assert.ThatBool(actual := view.Ready, message := "Ready must be false for STOPPED").IsFalse();
Assert.ThatBool(actual := view.Running, message := "Running must be false for STOPPED").IsFalse();
Assert.ThatBool(
	actual := view.StateChanged,
	message := "StateChanged must track its backing flag in STOPPED"
).IsFalse();
END_METHOD

//! <summary>Borrows the concrete class name. Callers must not modify the returned storage.</summary>
{attribute 'monitoring' := 'call'}
PROPERTY ClassName : REFERENCE TO STRING
GET
ClassName REF= _ClassName;
END_GET
END_PROPERTY

//! <summary>Borrows the compiler-initialized namespace name. Callers must not modify the returned storage.</summary>
{attribute 'monitoring' := 'call'}
PROPERTY NamespaceName : REFERENCE TO STRING
GET
NamespaceName REF= CurrentNamespace.Name;
END_GET
END_PROPERTY

//! <summary>Reports the complete concrete instance size in bytes.</summary>
{attribute 'monitoring' := 'call'}
PROPERTY SelfSize : ULINT
GET
SelfSize := XSIZEOF(THIS^);
END_GET
END_PROPERTY

END_FUNCTION_BLOCK

// ---- Tests/Tasks/UnboundTaskRunningSubstateTest.TcPOU
(*
SPDX-FileCopyrightText: © 2026 Oleksandr Tiutyk <trofimich@gmail.com>
SPDX-License-Identifier: MIT
License: https://opensource.org/license/mit
*)

(*!
<summary>Checks safe defaults for an unbound TaskRunningSubstate view.</summary>
<description>
Uses unbound local references and checks every observable property without dereferencing a missing target.
</description>
*)

{attribute 'no_explicit_call' := 'do not call this function block directly'}
FUNCTION_BLOCK UnboundTaskRunningSubstateTest EXTENDS TOF_Testing.SingleCycleTest
VAR_STAT
	{attribute 'hide'}
	_ClassName : STRING := __POUNAME();
END_VAR

//! <summary>Reads all flags and verifies the default value for an unbound view.</summary>
METHOD PROTECTED ExecuteTest
VAR
	backingValue : REFERENCE TO TOF_Tasks.TASK_RUNNING_SUBSTATE;
	view : TOF_Tasks.TaskRunningSubstate(taskRunningSubstate := backingValue);
END_VAR
Assert.ThatBool(
	actual := view.ResourceAcquiring,
	message := "Unbound TaskRunningSubstate.ResourceAcquiring must be false"
).IsFalse();
Assert.ThatBool(actual := view.Processing, message := "Unbound TaskRunningSubstate.Processing must be false").IsFalse();
Assert.ThatBool(actual := view.Stopping, message := "Unbound TaskRunningSubstate.Stopping must be false").IsFalse();
Assert.ThatBool(
	actual := view.ResourceReleasing,
	message := "Unbound TaskRunningSubstate.ResourceReleasing must be false"
).IsFalse();
Assert.ThatBool(
	actual := view.Value = TOF_Tasks.TASK_RUNNING_SUBSTATE.RESOURCE_ACQUIRING,
	message := "Unbound Value must default to RESOURCE_ACQUIRING"
).IsTrue();
END_METHOD

//! <summary>Borrows the concrete class name. Callers must not modify the returned storage.</summary>
{attribute 'monitoring' := 'call'}
PROPERTY ClassName : REFERENCE TO STRING
GET
ClassName REF= _ClassName;
END_GET
END_PROPERTY

//! <summary>Borrows the compiler-initialized namespace name. Callers must not modify the returned storage.</summary>
{attribute 'monitoring' := 'call'}
PROPERTY NamespaceName : REFERENCE TO STRING
GET
NamespaceName REF= CurrentNamespace.Name;
END_GET
END_PROPERTY

//! <summary>Reports the complete concrete instance size in bytes.</summary>
{attribute 'monitoring' := 'call'}
PROPERTY SelfSize : ULINT
GET
SelfSize := XSIZEOF(THIS^);
END_GET
END_PROPERTY

END_FUNCTION_BLOCK

// ---- Tests/Tasks/BoundTaskRunningSubstateTest.TcPOU
(*
SPDX-FileCopyrightText: © 2026 Oleksandr Tiutyk <trofimich@gmail.com>
SPDX-License-Identifier: MIT
License: https://opensource.org/license/mit
*)

(*!
<summary>Checks that a bound TaskRunningSubstate view observes changes to its backing data.</summary>
<description>
Exercises all defined values through the same view in one call. The backing data and view are local to the call.
</description>
*)

{attribute 'no_explicit_call' := 'do not call this function block directly'}
FUNCTION_BLOCK BoundTaskRunningSubstateTest EXTENDS TOF_Testing.SingleCycleTest
VAR_STAT
	{attribute 'hide'}
	_ClassName : STRING := __POUNAME();
END_VAR

//! <summary>Sets each backing value and checks the corresponding value and flags.</summary>
METHOD PROTECTED ExecuteTest
VAR
	backingValue : TOF_Tasks.TASK_RUNNING_SUBSTATE;
	view : TOF_Tasks.TaskRunningSubstate(taskRunningSubstate := backingValue);
END_VAR
backingValue := TOF_Tasks.TASK_RUNNING_SUBSTATE.RESOURCE_ACQUIRING;
Assert.ThatBool(
	actual := view.Value = TOF_Tasks.TASK_RUNNING_SUBSTATE.RESOURCE_ACQUIRING,
	message := "Value must track RESOURCE_ACQUIRING"
).IsTrue();
Assert.ThatBool(
	actual := view.ResourceAcquiring,
	message := "ResourceAcquiring must be true for RESOURCE_ACQUIRING"
).IsTrue();
Assert.ThatBool(actual := view.Processing, message := "Processing must be false for RESOURCE_ACQUIRING").IsFalse();
Assert.ThatBool(actual := view.Stopping, message := "Stopping must be false for RESOURCE_ACQUIRING").IsFalse();
Assert.ThatBool(
	actual := view.ResourceReleasing,
	message := "ResourceReleasing must be false for RESOURCE_ACQUIRING"
).IsFalse();

backingValue := TOF_Tasks.TASK_RUNNING_SUBSTATE.PROCESSING;
Assert.ThatBool(
	actual := view.Value = TOF_Tasks.TASK_RUNNING_SUBSTATE.PROCESSING,
	message := "Value must track PROCESSING"
).IsTrue();
Assert.ThatBool(actual := view.Processing, message := "Processing must be true for PROCESSING").IsTrue();
Assert.ThatBool(
	actual := view.ResourceAcquiring,
	message := "ResourceAcquiring must be false for PROCESSING"
).IsFalse();
Assert.ThatBool(actual := view.Stopping, message := "Stopping must be false for PROCESSING").IsFalse();
Assert.ThatBool(
	actual := view.ResourceReleasing,
	message := "ResourceReleasing must be false for PROCESSING"
).IsFalse();

backingValue := TOF_Tasks.TASK_RUNNING_SUBSTATE.STOPPING;
Assert.ThatBool(
	actual := view.Value = TOF_Tasks.TASK_RUNNING_SUBSTATE.STOPPING,
	message := "Value must track STOPPING"
).IsTrue();
Assert.ThatBool(actual := view.Stopping, message := "Stopping must be true for STOPPING").IsTrue();
Assert.ThatBool(actual := view.ResourceAcquiring, message := "ResourceAcquiring must be false for STOPPING").IsFalse();
Assert.ThatBool(actual := view.Processing, message := "Processing must be false for STOPPING").IsFalse();
Assert.ThatBool(actual := view.ResourceReleasing, message := "ResourceReleasing must be false for STOPPING").IsFalse();

backingValue := TOF_Tasks.TASK_RUNNING_SUBSTATE.RESOURCE_RELEASING;
Assert.ThatBool(
	actual := view.Value = TOF_Tasks.TASK_RUNNING_SUBSTATE.RESOURCE_RELEASING,
	message := "Value must track RESOURCE_RELEASING"
).IsTrue();
Assert.ThatBool(
	actual := view.ResourceReleasing,
	message := "ResourceReleasing must be true for RESOURCE_RELEASING"
).IsTrue();
Assert.ThatBool(
	actual := view.ResourceAcquiring,
	message := "ResourceAcquiring must be false for RESOURCE_RELEASING"
).IsFalse();
Assert.ThatBool(actual := view.Processing, message := "Processing must be false for RESOURCE_RELEASING").IsFalse();
Assert.ThatBool(actual := view.Stopping, message := "Stopping must be false for RESOURCE_RELEASING").IsFalse();
END_METHOD

//! <summary>Borrows the concrete class name. Callers must not modify the returned storage.</summary>
{attribute 'monitoring' := 'call'}
PROPERTY ClassName : REFERENCE TO STRING
GET
ClassName REF= _ClassName;
END_GET
END_PROPERTY

//! <summary>Borrows the compiler-initialized namespace name. Callers must not modify the returned storage.</summary>
{attribute 'monitoring' := 'call'}
PROPERTY NamespaceName : REFERENCE TO STRING
GET
NamespaceName REF= CurrentNamespace.Name;
END_GET
END_PROPERTY

//! <summary>Reports the complete concrete instance size in bytes.</summary>
{attribute 'monitoring' := 'call'}
PROPERTY SelfSize : ULINT
GET
SelfSize := XSIZEOF(THIS^);
END_GET
END_PROPERTY

END_FUNCTION_BLOCK

// ---- Tests/Tasks/UnboundTaskStopReasonTest.TcPOU
(*
SPDX-FileCopyrightText: © 2026 Oleksandr Tiutyk <trofimich@gmail.com>
SPDX-License-Identifier: MIT
License: https://opensource.org/license/mit
*)

(*!
<summary>Checks safe defaults for an unbound TaskStopReason view.</summary>
<description>
Uses unbound local references and checks every observable property without dereferencing a missing target.
</description>
*)

{attribute 'no_explicit_call' := 'do not call this function block directly'}
FUNCTION_BLOCK UnboundTaskStopReasonTest EXTENDS TOF_Testing.SingleCycleTest
VAR_STAT
	{attribute 'hide'}
	_ClassName : STRING := __POUNAME();
END_VAR

//! <summary>Reads all flags and verifies the default value for an unbound view.</summary>
METHOD PROTECTED ExecuteTest
VAR
	backingValue : REFERENCE TO TOF_Tasks.TASK_STOP_REASON;
	stopMessage : REFERENCE TO TOF_Core.ERROR_MESSAGE;
	view : TOF_Tasks.TaskStopReason(stopReason := backingValue, stopReasonMessage := stopMessage);
END_VAR
Assert.ThatBool(actual := view.WorkDone, message := "Unbound TaskStopReason.WorkDone must be false").IsFalse();
Assert.ThatBool(actual := view.Failure, message := "Unbound TaskStopReason.Failure must be false").IsFalse();
Assert.ThatBool(
	actual := view.ExternalCancel,
	message := "Unbound TaskStopReason.ExternalCancel must be false"
).IsFalse();
Assert.ThatBool(
	actual := view.InternalAbort,
	message := "Unbound TaskStopReason.InternalAbort must be false"
).IsFalse();
Assert.ThatBool(
	actual := view.Value = TOF_Tasks.TASK_STOP_REASON.WORK_DONE,
	message := "Unbound Value must default to WORK_DONE"
).IsTrue();
Assert.ThatBool(
	actual := __ISVALIDREF(view.Message),
	message := "Unbound stop message reference must be invalid"
).IsFalse();
END_METHOD

//! <summary>Borrows the concrete class name. Callers must not modify the returned storage.</summary>
{attribute 'monitoring' := 'call'}
PROPERTY ClassName : REFERENCE TO STRING
GET
ClassName REF= _ClassName;
END_GET
END_PROPERTY

//! <summary>Borrows the compiler-initialized namespace name. Callers must not modify the returned storage.</summary>
{attribute 'monitoring' := 'call'}
PROPERTY NamespaceName : REFERENCE TO STRING
GET
NamespaceName REF= CurrentNamespace.Name;
END_GET
END_PROPERTY

//! <summary>Reports the complete concrete instance size in bytes.</summary>
{attribute 'monitoring' := 'call'}
PROPERTY SelfSize : ULINT
GET
SelfSize := XSIZEOF(THIS^);
END_GET
END_PROPERTY

END_FUNCTION_BLOCK

// ---- Tests/Tasks/BoundTaskStopReasonTest.TcPOU
(*
SPDX-FileCopyrightText: © 2026 Oleksandr Tiutyk <trofimich@gmail.com>
SPDX-License-Identifier: MIT
License: https://opensource.org/license/mit
*)

(*!
<summary>Checks that a bound TaskStopReason view observes changes to its backing data.</summary>
<description>
Exercises all defined values through the same view in one call. The backing data and view are local to the call.
</description>
*)

{attribute 'no_explicit_call' := 'do not call this function block directly'}
FUNCTION_BLOCK BoundTaskStopReasonTest EXTENDS TOF_Testing.SingleCycleTest
VAR_STAT
	{attribute 'hide'}
	_ClassName : STRING := __POUNAME();
END_VAR

//! <summary>Sets each backing value and checks the corresponding value and flags.</summary>
METHOD PROTECTED ExecuteTest
VAR
	backingValue : TOF_Tasks.TASK_STOP_REASON;
	stopMessage : TOF_Core.ERROR_MESSAGE;
	view : TOF_Tasks.TaskStopReason(stopReason := backingValue, stopReasonMessage := stopMessage);
END_VAR
backingValue := TOF_Tasks.TASK_STOP_REASON.WORK_DONE;
stopMessage := "initial message";
Assert.ThatBool(
	actual := view.Value = TOF_Tasks.TASK_STOP_REASON.WORK_DONE,
	message := "Value must track WORK_DONE"
).IsTrue();
Assert.ThatBool(actual := view.WorkDone, message := "WorkDone must be true for WORK_DONE").IsTrue();
Assert.ThatBool(actual := view.Failure, message := "Failure must be false for WORK_DONE").IsFalse();
Assert.ThatBool(actual := view.ExternalCancel, message := "ExternalCancel must be false for WORK_DONE").IsFalse();
Assert.ThatBool(actual := view.InternalAbort, message := "InternalAbort must be false for WORK_DONE").IsFalse();
Assert.ThatBool(actual := __ISVALIDREF(view.Message), message := "Message must be bound for WORK_DONE").IsTrue();

IF __ISVALIDREF(view.Message) THEN
	Assert.ThatBool(
		actual := view.Message = "initial message",
		message := "Message must match the backing text for WORK_DONE"
	).IsTrue();
END_IF

backingValue := TOF_Tasks.TASK_STOP_REASON.FAILURE;
stopMessage := "diagnostic failure";
Assert.ThatBool(
	actual := view.Value = TOF_Tasks.TASK_STOP_REASON.FAILURE,
	message := "Value must track FAILURE"
).IsTrue();
Assert.ThatBool(actual := view.Failure, message := "Failure must be true for FAILURE").IsTrue();
Assert.ThatBool(actual := view.WorkDone, message := "WorkDone must be false for FAILURE").IsFalse();
Assert.ThatBool(actual := view.ExternalCancel, message := "ExternalCancel must be false for FAILURE").IsFalse();
Assert.ThatBool(actual := view.InternalAbort, message := "InternalAbort must be false for FAILURE").IsFalse();
Assert.ThatBool(actual := __ISVALIDREF(view.Message), message := "Message must be bound for FAILURE").IsTrue();

IF __ISVALIDREF(view.Message) THEN
	Assert.ThatBool(
		actual := view.Message = "diagnostic failure",
		message := "Message must match the backing text for FAILURE"
	).IsTrue();
END_IF

backingValue := TOF_Tasks.TASK_STOP_REASON.EXTERNAL_CANCEL;
Assert.ThatBool(
	actual := view.Value = TOF_Tasks.TASK_STOP_REASON.EXTERNAL_CANCEL,
	message := "Value must track EXTERNAL_CANCEL"
).IsTrue();
Assert.ThatBool(actual := view.ExternalCancel, message := "ExternalCancel must be true for EXTERNAL_CANCEL").IsTrue();
Assert.ThatBool(actual := view.WorkDone, message := "WorkDone must be false for EXTERNAL_CANCEL").IsFalse();
Assert.ThatBool(actual := view.Failure, message := "Failure must be false for EXTERNAL_CANCEL").IsFalse();
Assert.ThatBool(actual := view.InternalAbort, message := "InternalAbort must be false for EXTERNAL_CANCEL").IsFalse();

backingValue := TOF_Tasks.TASK_STOP_REASON.INTERNAL_ABORT;
Assert.ThatBool(
	actual := view.Value = TOF_Tasks.TASK_STOP_REASON.INTERNAL_ABORT,
	message := "Value must track INTERNAL_ABORT"
).IsTrue();
Assert.ThatBool(actual := view.InternalAbort, message := "InternalAbort must be true for INTERNAL_ABORT").IsTrue();
Assert.ThatBool(actual := view.WorkDone, message := "WorkDone must be false for INTERNAL_ABORT").IsFalse();
Assert.ThatBool(actual := view.Failure, message := "Failure must be false for INTERNAL_ABORT").IsFalse();
Assert.ThatBool(actual := view.ExternalCancel, message := "ExternalCancel must be false for INTERNAL_ABORT").IsFalse();
END_METHOD

//! <summary>Borrows the concrete class name. Callers must not modify the returned storage.</summary>
{attribute 'monitoring' := 'call'}
PROPERTY ClassName : REFERENCE TO STRING
GET
ClassName REF= _ClassName;
END_GET
END_PROPERTY

//! <summary>Borrows the compiler-initialized namespace name. Callers must not modify the returned storage.</summary>
{attribute 'monitoring' := 'call'}
PROPERTY NamespaceName : REFERENCE TO STRING
GET
NamespaceName REF= CurrentNamespace.Name;
END_GET
END_PROPERTY

//! <summary>Reports the complete concrete instance size in bytes.</summary>
{attribute 'monitoring' := 'call'}
PROPERTY SelfSize : ULINT
GET
SelfSize := XSIZEOF(THIS^);
END_GET
END_PROPERTY

END_FUNCTION_BLOCK

// ---- Tests/Tasks/TaskReinitViewsTest.TcPOU
(*
SPDX-FileCopyrightText: © 2026 Oleksandr Tiutyk <trofimich@gmail.com>
SPDX-License-Identifier: MIT
License: https://opensource.org/license/mit
*)

(*!
<summary>Checks that reinitialization preserves a task's live views while cancellation is pending.</summary>
<description>
Exercises the reinitialization hook in place on a resource-free task. Copy-code relocation requires a runtime check.
</description>
*)

{attribute 'no_explicit_call' := 'do not call this function block directly'}
FUNCTION_BLOCK TaskReinitViewsTest EXTENDS TOF_Testing.SingleCycleTest
VAR_STAT
	{attribute 'hide'}
	_ClassName : STRING := __POUNAME();
END_VAR

//! <summary>Requests cancellation, calls FB_reinit in STOPPING and observes the original and final stop diagnostics.</summary>
METHOD PROTECTED ExecuteTest
VAR
	task : CounterTask(name := "Reinit view fixture");
	started : BOOL;
	cancelled : BOOL;
	reinitialized : BOOL;
END_VAR
Assert.ThatBool(actual := task.State.Ready, message := "Task must begin in READY").IsTrue();
Assert.ThatBool(actual := task.FinalStopReason.WorkDone, message := "Initial final reason must be WORK_DONE").IsTrue();

started := task.Start();
Assert.ThatBool(actual := started, message := "Fixture must accept Start").IsTrue();

IF NOT started THEN
	RETURN;
END_IF

Assert.ThatBool(
	actual := task.RunningSubstate.Processing,
	message := "Resource-free task must start in PROCESSING"
).IsTrue();
cancelled := task.Cancel();
Assert.ThatBool(actual := cancelled, message := "Fixture must accept Cancel").IsTrue();

IF NOT cancelled THEN
	RETURN;
END_IF

reinitialized := task.FB_reinit();
Assert.ThatBool(actual := reinitialized, message := "FB_reinit must return true").IsTrue();
Assert.ThatBool(
	actual := task.State.Running,
	message := "Reinitialization must preserve RUNNING during cancellation"
).IsTrue();
Assert.ThatBool(
	actual := task.State.StateChanged,
	message := "Reinitialization must preserve the lifecycle transition flag"
).IsTrue();
Assert.ThatBool(
	actual := task.RunningSubstate.Stopping,
	message := "Reinitialization must preserve the STOPPING phase"
).IsTrue();
Assert.ThatBool(
	actual := task.OriginalStopReason.ExternalCancel,
	message := "Reinitialization must preserve the requested cancellation"
).IsTrue();
Assert.ThatBool(
	actual := __ISVALIDREF(task.OriginalStopReason.Message),
	message := "Original cancellation diagnostic must be bound"
).IsTrue();

IF __ISVALIDREF(task.OriginalStopReason.Message) THEN
	Assert.ThatBool(
		actual := task.OriginalStopReason.Message = "Cancelled by external logic",
		message := "Reinitialization must preserve the original cancellation diagnostic"
	).IsTrue();
END_IF

task.Execute();
Assert.ThatBool(
	actual := task.State.Stopped,
	message := "The state view must observe completion of cancellation"
).IsTrue();
Assert.ThatBool(
	actual := task.FinalStopReason.ExternalCancel,
	message := "The final reason view must observe the completed cancellation"
).IsTrue();
Assert.ThatBool(
	actual := __ISVALIDREF(task.FinalStopReason.Message),
	message := "Final cancellation diagnostic must be bound"
).IsTrue();

IF __ISVALIDREF(task.FinalStopReason.Message) THEN
	Assert.ThatBool(
		actual := task.FinalStopReason.Message = "Cancelled by external logic",
		message := "The final message view must observe the copied cancellation diagnostic"
	).IsTrue();
END_IF
END_METHOD

//! <summary>Borrows the concrete class name. Callers must not modify the returned storage.</summary>
{attribute 'monitoring' := 'call'}
PROPERTY ClassName : REFERENCE TO STRING
GET
ClassName REF= _ClassName;
END_GET
END_PROPERTY

//! <summary>Borrows the compiler-initialized namespace name. Callers must not modify the returned storage.</summary>
{attribute 'monitoring' := 'call'}
PROPERTY NamespaceName : REFERENCE TO STRING
GET
NamespaceName REF= CurrentNamespace.Name;
END_GET
END_PROPERTY

//! <summary>Reports the complete concrete instance size in bytes.</summary>
{attribute 'monitoring' := 'call'}
PROPERTY SelfSize : ULINT
GET
SelfSize := XSIZEOF(THIS^);
END_GET
END_PROPERTY

END_FUNCTION_BLOCK

// ---- Tests/Tasks/Sequence/CounterTask.TcPOU
(*
SPDX-FileCopyrightText: © 2026 Oleksandr Tiutyk <trofimich@gmail.com>
SPDX-License-Identifier: MIT
License: https://opensource.org/license/mit
*)

(*!
<summary>Provides a resource-free task that counts one step per work call.</summary>
<description>
Configure the target before Start. A successful Reset from STOPPED clears the counter and retains the target.
</description>
*)

FUNCTION_BLOCK CounterTask EXTENDS TOF_Tasks.Task
VAR_STAT
	//! <summary>Class name shared by all instances of this function block.</summary>
	{attribute 'hide'} 
	_ClassName : STRING := __POUNAME();
END_VAR
VAR
	_Counter : INT;
	_TargetValue : INT;
END_VAR

{attribute 'monitoring' := 'call'}
PROPERTY ClassName : REFERENCE TO STRING
GET
ClassName REF= _ClassName;
END_GET
END_PROPERTY

{attribute 'monitoring' := 'call'}
PROPERTY Counter : INT
GET
Counter := _Counter;
END_GET
END_PROPERTY

{attribute 'monitoring' := 'call'}
PROPERTY NamespaceName : REFERENCE TO STRING
GET
NamespaceName REF= CurrentNamespace.Name;
END_GET
END_PROPERTY

METHOD PROTECTED OnRunning
VAR_OUTPUT
	processingState : TOF_Tasks.TASK_PROCESSING_STATE;
END_VAR
VAR_IN_OUT
	stopReasonMessage : TOF_Core.ERROR_MESSAGE;
END_VAR
_Counter := _Counter + 1;

IF _Counter >= _TargetValue THEN
	processingState := TOF_Tasks.TASK_PROCESSING_STATE.DONE;
END_IF
END_METHOD

(*!
<summary>Clears progress for a stopped counter while retaining its configured target.</summary>
<description>
Invoked by Task.Reset after termination. A counter prepared for the next run starts from zero.
</description>
*)
METHOD PROTECTED OnReset
_Counter := TOF_Core.SignedInt16.ZERO;
END_METHOD

{attribute 'monitoring' := 'call'}
PROPERTY SelfSize : ULINT
GET
SelfSize := XSIZEOF(THIS^);
END_GET
END_PROPERTY

{attribute 'monitoring' := 'call'}
PROPERTY TargetValue : INT
GET
TargetValue := _TargetValue;
END_GET
SET
_TargetValue := TargetValue;
END_SET
END_PROPERTY

END_FUNCTION_BLOCK

// ---- Tests/Tasks/TaskNamePreservedByResetTest.TcPOU
(*
SPDX-FileCopyrightText: © 2026 Oleksandr Tiutyk <trofimich@gmail.com>
SPDX-License-Identifier: MIT
License: https://opensource.org/license/mit
*)

(*!
<summary>Checks that a configured task name survives the STOPPED to READY reset.</summary>
<description>
Completes a resource-free one-step task before invoking Reset. A new local fixture is used on every run.
</description>
*)

{attribute 'no_explicit_call' := 'do not call this function block directly'}
FUNCTION_BLOCK TaskNamePreservedByResetTest EXTENDS TOF_Testing.SingleCycleTest
VAR_STAT
	{attribute 'hide'}
	_ClassName : STRING := __POUNAME();
END_VAR

//! <summary>Verifies the constructor name and exercises Reset from STOPPED before checking that name again.</summary>
METHOD PROTECTED ExecuteTest
VAR
	task : CounterTask(name := "Configured counter");
	started : BOOL;
	resetSucceeded : BOOL;
END_VAR
Assert.ThatWideString(actual := task.Name, message := "Task must adopt the explicit constructor name")
	.ToBe(expected := "Configured counter");

task.TargetValue := 1;
started := task.Start();
Assert.ThatBool(actual := started, message := "Fixture must accept Start").IsTrue();

IF NOT started THEN
	RETURN;
END_IF

task.Execute();
Assert.ThatBool(actual := task.State.Stopped, message := "Reset test requires a completed task").IsTrue();

IF NOT task.State.Stopped THEN
	RETURN;
END_IF

resetSucceeded := task.Reset();
Assert.ThatBool(actual := resetSucceeded, message := "Fixture must accept Reset from STOPPED").IsTrue();
Assert.ThatBool(actual := task.State.Ready, message := "Reset must return the fixture to READY").IsTrue();
Assert.ThatWideString(actual := task.Name, message := "Reset from STOPPED must preserve the configured name")
	.ToBe(expected := "Configured counter");
END_METHOD

//! <summary>Borrows the concrete class name. Callers must not modify the returned storage.</summary>
{attribute 'monitoring' := 'call'}
PROPERTY ClassName : REFERENCE TO STRING
GET
ClassName REF= _ClassName;
END_GET
END_PROPERTY

//! <summary>Borrows the compiler-initialized namespace name. Callers must not modify the returned storage.</summary>
{attribute 'monitoring' := 'call'}
PROPERTY NamespaceName : REFERENCE TO STRING
GET
NamespaceName REF= CurrentNamespace.Name;
END_GET
END_PROPERTY

//! <summary>Reports the complete concrete instance size in bytes.</summary>
{attribute 'monitoring' := 'call'}
PROPERTY SelfSize : ULINT
GET
SelfSize := XSIZEOF(THIS^);
END_GET
END_PROPERTY

END_FUNCTION_BLOCK

// ---- Tests/Tasks/Sequence/TaskSequenceTestGroup.TcPOU
(*
SPDX-FileCopyrightText: © 2026 Oleksandr Tiutyk <trofimich@gmail.com>
SPDX-License-Identifier: MIT
License: https://opensource.org/license/mit
*)

(*!
<summary>Groups the cyclic FIFO and both empty-queue modes.</summary>
<description>
Owns three cases and their fixed registration array. Use the group from one task and keep it at a stable address.
</description>
*)

{attribute 'no_assign'}
{attribute 'no_explicit_call' := 'do not call this function block directly'}
FUNCTION_BLOCK TaskSequenceTestGroup EXTENDS TOF_Testing.TestGroup<3>
VAR_STAT
	{attribute 'hide'}
	_ClassName : STRING := __POUNAME();
END_VAR
VAR
	_Sequence : TaskSequenceFifoTest(name := "TestSequence", parent := THIS^);
	_AutomaticStop : TaskQueueEmptyModeTest(
		name := "StopWhenNoPendingTasksEnabled",
		parent := THIS^,
		stopWhenEmpty := TRUE
	);
	_WaitForWork : TaskQueueEmptyModeTest(
		name := "StopWhenNoPendingTasksDisabled",
		parent := THIS^,
		stopWhenEmpty := FALSE
	);

	_Children : ARRAY [0.._ChildCount - 1] OF TOF_Testing.ITestElement :=
	[
		_Sequence,
		_AutomaticStop,
		_WaitForWork
	];
END_VAR

//! <summary>Borrows the fixed child array. Callers must not modify it.</summary>
{attribute 'monitoring' := 'call'}
PROPERTY Children : REFERENCE TO ARRAY [0.._ChildCount - 1] OF TOF_Testing.ITestElement
GET
Children REF= _Children;
END_GET
END_PROPERTY

//! <summary>Borrows the concrete class name. Callers must not modify the returned storage.</summary>
{attribute 'monitoring' := 'call'}
PROPERTY ClassName : REFERENCE TO STRING
GET
ClassName REF= _ClassName;
END_GET
END_PROPERTY

//! <summary>Borrows the compiler-initialized namespace name. Callers must not modify it.</summary>
{attribute 'monitoring' := 'call'}
PROPERTY NamespaceName : REFERENCE TO STRING
GET
NamespaceName REF= CurrentNamespace.Name;
END_GET
END_PROPERTY

//! <summary>Reports the complete concrete instance size in bytes.</summary>
{attribute 'monitoring' := 'call'}
PROPERTY SelfSize : ULINT
GET
SelfSize := XSIZEOF(THIS^);
END_GET
END_PROPERTY

END_FUNCTION_BLOCK

// ---- Tests/Tasks/Sequence/TaskSequenceFifoTest.TcPOU
(*
SPDX-FileCopyrightText: © 2026 Oleksandr Tiutyk <trofimich@gmail.com>
SPDX-License-Identifier: MIT
License: https://opensource.org/license/mit
*)

(*!
<summary>Checks FIFO dispatch and one child step per PLC cycle.</summary>
<description>
Owns a reusable queue that borrows three counters with no external resources. Use in one task.
Copying would invalidate internal references and queue ownership.
</description>
*)

{attribute 'no_assign'}
{attribute 'no_explicit_call' := 'do not call this function block directly'}
FUNCTION_BLOCK TaskSequenceFifoTest EXTENDS TOF_Testing.MultiCycleTest
VAR_STAT
	{attribute 'hide'}
	_ClassName : STRING := __POUNAME();
END_VAR
VAR CONSTANT
	//! <summary>Step counts for the three resource-free children.</summary>
	_FirstTarget : INT := 2;
	_SecondTarget : INT := 3;
	_ThirdTarget : INT := 4;

	//! <summary>Each start uses one call, then each work step uses a separate call.</summary>
	_FirstStartCycle : INT := 1;
	_FirstFinishCycle : INT := _FirstStartCycle + _FirstTarget;
	_SecondStartCycle : INT := _FirstFinishCycle + 1;
	_SecondFinishCycle : INT := _SecondStartCycle + _SecondTarget;
	_ThirdStartCycle : INT := _SecondFinishCycle + 1;
	_ThirdFinishCycle : INT := _ThirdStartCycle + _ThirdTarget;
END_VAR
VAR
	_Queue : TOF_Tasks.StandardTaskQueue(name := "FIFO test queue");
	_First : CounterTask(name := "First child");
	_Second : CounterTask(name := "Second child");
	_Third : CounterTask(name := "Third child");
END_VAR

(*!
<summary>Enqueues three READY children and starts the queue without executing any child.</summary>
*)
METHOD PROTECTED BeforeTest
IF NOT _Queue.State.Ready
	OR_ELSE _Queue.PendingTaskCount <> 0
	OR_ELSE NOT _First.State.Ready
	OR_ELSE NOT _Second.State.Ready
	OR_ELSE NOT _Third.State.Ready
THEN
	RecordFailure(message := "FIFO test requires an empty READY queue and three READY children");
	RETURN;
END_IF

Assert.ThatBool(
	actual := _Queue.StopWhenNoPendingTasks,
	message := "The queue must default to waiting when empty"
).IsFalse();

_First.TargetValue := _FirstTarget;
_Second.TargetValue := _SecondTarget;
_Third.TargetValue := _ThirdTarget;

_Queue.Enqueue(task := _First);
_Queue.Enqueue(task := _Second);
_Queue.Enqueue(task := _Third);

Assert.ThatDInt(
	actual := _Queue.PendingTaskCount,
	message := "Queue must retain all three entries"
).ToBe(expected := 3);
Assert.ThatBool(actual := _Queue.Start(), message := "Prepared FIFO queue must accept Start").IsTrue();
END_METHOD

(*!
<summary>Checks one queue call per PLC cycle against the expected order and progress.</summary>
<description>
Requests cancellation after the last removal and observes the stopped queue in the following cycle.
</description>
*)
METHOD PROTECTED ExecuteTest : TOF_Testing.TEST_CYCLE_RESULT
VAR
	cycle : INT;
	expectedPending : DINT;
END_VAR
ExecuteTest := TOF_Testing.TEST_CYCLE_RESULT.DONE;
cycle := TO_INT(CycleCount);
_Queue.Execute();

IF cycle > _ThirdFinishCycle THEN
	Assert.ThatBool(actual := _Queue.State.Stopped, message := "Empty queue must stop after Cancel").IsTrue();
	Assert.ThatBool(
		actual := _Queue.FinalStopReason.ExternalCancel,
		message := "The completed FIFO run must end with external cancellation"
	).IsTrue();

	RETURN;
END_IF

checkChild(child := _First, startCycle := _FirstStartCycle, target := _FirstTarget, cycle := cycle);
checkChild(child := _Second, startCycle := _SecondStartCycle, target := _SecondTarget, cycle := cycle);
checkChild(child := _Third, startCycle := _ThirdStartCycle, target := _ThirdTarget, cycle := cycle);

IF cycle >= _ThirdFinishCycle THEN
	expectedPending := 0;
ELSIF cycle >= _SecondFinishCycle THEN
	expectedPending := 1;
ELSIF cycle >= _FirstFinishCycle THEN
	expectedPending := 2;
ELSE
	expectedPending := 3;
END_IF

Assert.ThatDInt(
	actual := _Queue.PendingTaskCount,
	message := "Pending count must include the current child until successful completion"
).ToBe(expected := expectedPending);
Assert.ThatBool(actual := _Queue.State.Running, message := "FIFO queue must keep running until Cancel").IsTrue();

IF cycle = _ThirdFinishCycle THEN
	Assert.ThatBool(actual := _Queue.Cancel(), message := "Drained FIFO queue must accept Cancel").IsTrue();
END_IF

ExecuteTest := TOF_Testing.TEST_CYCLE_RESULT.BUSY;
END_METHOD

(*!
<summary>Checks a child's position and progress on the expected schedule.</summary>
<description>
Observes the borrowed child without driving it. The start call performs zero work steps.
</description>
<param name="child">Live counter to observe.</param>
<param name="startCycle">First queue call allowed to start this child.</param>
<param name="target">Number of work steps required to complete the child.</param>
<param name="cycle">Current test cycle.</param>
*)
METHOD PRIVATE checkChild
VAR_INPUT
	child : REFERENCE TO CounterTask;
	startCycle : INT;
	target : INT;
	cycle : INT;
END_VAR
VAR
	elapsedSteps : INT;
END_VAR
elapsedSteps := cycle - startCycle;
Assert.ThatInt(
	actual := child.Counter,
	message := TOF_Core.WideStrings.ConcatFit255(child.Name, " must advance one step per work call")
).ToBe(expected := LIMIT(TOF_Core.SignedInt16.ZERO, elapsedSteps, target));

IF cycle < startCycle THEN
	Assert.ThatBool(
		actual := child.State.Ready,
		message := TOF_Core.WideStrings.ConcatFit255(child.Name, " must wait in READY until its turn")
	).IsTrue();
ELSIF elapsedSteps < target THEN
	Assert.ThatBool(
		actual := child.State.Running,
		message := TOF_Core.WideStrings.ConcatFit255(child.Name, " must be RUNNING during its turn")
	).IsTrue();
ELSE
	Assert.ThatBool(
		actual := child.State.Stopped AND_THEN child.FinalStopReason.WorkDone,
		message := TOF_Core.WideStrings.ConcatFit255(child.Name, " must be STOPPED with WorkDone after its last step")
	).IsTrue();
END_IF
END_METHOD

(*!
<summary>Stops and empties the queue before resetting its former children.</summary>
<description>
Checks that the resource-free fixture can finish cancellation in one call. If the queue is still running,
reports cleanup failure and leaves its children under queue control.
</description>
*)
METHOD PROTECTED AfterTest
IF _Queue.State.Running THEN
	IF _Queue.OriginalStopReason.ExternalCancel OR_ELSE _Queue.Cancel() THEN
		_Queue.Execute();
	END_IF
END_IF

IF _Queue.State.Running THEN
	RecordFailure(message := "Cleanup could not stop the queue");
	RETURN;
END_IF

IF _Queue.State.Stopped THEN
	IF NOT _Queue.Reset() THEN
		RecordFailure(message := "Stopped queue refused Reset during cleanup");
		RETURN;
	END_IF
ELSE
	_Queue.ClearWaitingTasks();
END_IF

IF NOT _Queue.State.Ready OR_ELSE _Queue.PendingTaskCount <> 0 THEN
	RecordFailure(message := "Queue must be READY and empty before resetting its former children");
	RETURN;
END_IF

Assert.ThatBool(actual := _First.Reset(), message := "First child must accept cleanup Reset").IsTrue();
Assert.ThatBool(actual := _Second.Reset(), message := "Second child must accept cleanup Reset").IsTrue();
Assert.ThatBool(actual := _Third.Reset(), message := "Third child must accept cleanup Reset").IsTrue();
END_METHOD

//! <summary>Borrows the concrete class name. Callers must not modify the returned storage.</summary>
{attribute 'monitoring' := 'call'}
PROPERTY ClassName : REFERENCE TO STRING
GET
ClassName REF= _ClassName;
END_GET
END_PROPERTY

//! <summary>Borrows the compiler-initialized namespace name. Callers must not modify it.</summary>
{attribute 'monitoring' := 'call'}
PROPERTY NamespaceName : REFERENCE TO STRING
GET
NamespaceName REF= CurrentNamespace.Name;
END_GET
END_PROPERTY

//! <summary>Reports the complete concrete instance size in bytes.</summary>
{attribute 'monitoring' := 'call'}
PROPERTY SelfSize : ULINT
GET
SelfSize := XSIZEOF(THIS^);
END_GET
END_PROPERTY

END_FUNCTION_BLOCK

// ---- Tests/Tasks/Sequence/TaskQueueEmptyModeTest.TcPOU
(*
SPDX-FileCopyrightText: © 2026 Oleksandr Tiutyk <trofimich@gmail.com>
SPDX-License-Identifier: MIT
License: https://opensource.org/license/mit
*)

(*!
<summary>Checks one setting of StopWhenNoPendingTasks for empty and populated queues.</summary>
<description>
Owns separate resource-free fixtures per case. Calls Execute a bounded number of times in one task cycle.
Copying would invalidate internal references and queue ownership.
</description>
*)

{attribute 'no_assign'}
{attribute 'no_explicit_call' := 'do not call this function block directly'}
FUNCTION_BLOCK TaskQueueEmptyModeTest EXTENDS TOF_Testing.SingleCycleTest
VAR_STAT
	{attribute 'hide'}
	_ClassName : STRING := __POUNAME();
END_VAR
VAR CONSTANT
	//! <summary>Number of work calls needed by the counter after its separate start call.</summary>
	_Target : INT := 3;
END_VAR
VAR
	_StopWhenEmpty : BOOL;
	_Queue : TOF_Tasks.StandardTaskQueue(name := "Empty mode queue");
	_Child : CounterTask(name := "Empty mode child");
END_VAR

(*!
<summary>Stores the queue mode selected by this case.</summary>
<param name="name">Display name of this case.</param>
<param name="parent">Group that owns this case.</param>
<param name="stopWhenEmpty">TRUE tests automatic completion. FALSE tests waiting and late enqueue.</param>
*)
METHOD FB_init : BOOL
VAR_INPUT
	bInitRetains: BOOL; // TRUE: the retain variables are initialized (reset warm / reset cold)
	bInCopyCode: BOOL; // TRUE: the instance will be copied to the copy code afterward (online change)
	name : WSTRING;
	parent : TOF_Testing.ITestElement;
	stopWhenEmpty : BOOL;
END_VAR
_StopWhenEmpty := stopWhenEmpty;
FB_init := TRUE;
END_METHOD

(*!
<summary>Exercises an empty queue, then a completed child under the same mode.</summary>
<description>
With automatic completion, restarts the empty stopped queue with a prepared child. Otherwise adds the
child to the running empty queue, verifies that it can wait again, and explicitly cancels.
</description>
*)
METHOD PROTECTED ExecuteTest
VAR
	i : INT;
END_VAR
IF NOT _Queue.State.Ready OR_ELSE _Queue.PendingTaskCount <> 0 OR_ELSE NOT _Child.State.Ready THEN
	RecordFailure(message := "Empty mode test requires an empty READY queue and a READY child");
	RETURN;
END_IF

_Queue.StopWhenNoPendingTasks := _StopWhenEmpty;

IF NOT _Queue.Start() THEN
	RecordFailure(message := "An empty READY queue must accept Start");
	RETURN;
END_IF

_Queue.Execute();

IF _StopWhenEmpty THEN
	IF NOT _Queue.State.Stopped THEN
		RecordFailure(message := "Automatic mode must stop the initially empty queue");
		RETURN;
	END_IF

	Assert.ThatBool(
		actual := _Queue.FinalStopReason.WorkDone,
		message := "Initially empty queue must finish with WorkDone"
	).IsTrue();

	IF NOT _Queue.Reset() THEN
		RecordFailure(message := "Initially empty queue must accept Reset after completion");
		RETURN;
	END_IF

	_Queue.StopWhenNoPendingTasks := TRUE;
ELSIF NOT _Queue.State.Running THEN
	RecordFailure(message := "Waiting mode must keep the initially empty queue running");
	RETURN;
END_IF

_Child.TargetValue := _Target;
_Queue.Enqueue(task := _Child);
Assert.ThatDInt(actual := _Queue.PendingTaskCount, message := "Queue must retain the new child").ToBe(expected := 1);

IF _StopWhenEmpty AND_THEN NOT _Queue.Start() THEN
	RecordFailure(message := "READY queue with a prepared child must accept Start");
	RETURN;
END_IF

_Queue.Execute();

FOR i := 1 TO _Target DO
	_Queue.Execute();
END_FOR

Assert.ThatInt(actual := _Child.Counter, message := "The enqueued child must finish exactly its work")
	.ToBe(expected := _Target);
Assert.ThatBool(
	actual := _Child.State.Stopped AND_THEN _Child.FinalStopReason.WorkDone,
	message := "The enqueued child must finish in STOPPED with WorkDone"
).IsTrue();
Assert.ThatDInt(
	actual := _Queue.PendingTaskCount,
	message := "The successfully completed child must be removed"
).ToBe(expected := 0);
Assert.ThatBool(
	actual := _Queue.State.Running,
	message := "The last child must be removed before the queue handles the empty state"
).IsTrue();

_Queue.Execute();

IF _StopWhenEmpty THEN
	Assert.ThatBool(
		actual := _Queue.State.Stopped AND_THEN _Queue.FinalStopReason.WorkDone,
		message := "Automatic mode must stop with WorkDone when the last child has been removed"
	).IsTrue();

	RETURN;
END_IF

Assert.ThatBool(
	actual := _Queue.State.Running,
	message := "Waiting mode must remain running after the last child has been removed"
).IsTrue();

IF NOT _Queue.Cancel() THEN
	RecordFailure(message := "The empty running queue must accept Cancel");
	RETURN;
END_IF

_Queue.Execute();
Assert.ThatBool(
	actual := _Queue.State.Stopped AND_THEN _Queue.FinalStopReason.ExternalCancel,
	message := "The empty queue must stop with ExternalCancel after accepted cancellation"
).IsTrue();
END_METHOD

(*!
<summary>Stops and empties the queue before resetting its counter.</summary>
<description>
Checks for completion after one cancellation call to Execute. Leaves a still-running queue in control of its child.
</description>
*)
METHOD PROTECTED AfterTest
IF _Queue.State.Running THEN
	IF _Queue.OriginalStopReason.ExternalCancel OR_ELSE _Queue.Cancel() THEN
		_Queue.Execute();
	END_IF
END_IF

IF _Queue.State.Running THEN
	RecordFailure(message := "Cleanup could not stop the queue");
	RETURN;
END_IF

IF _Queue.State.Stopped THEN
	IF NOT _Queue.Reset() THEN
		RecordFailure(message := "Stopped queue refused Reset during cleanup");
		RETURN;
	END_IF
ELSE
	_Queue.ClearWaitingTasks();
END_IF

IF NOT _Queue.State.Ready OR_ELSE _Queue.PendingTaskCount <> 0 THEN
	RecordFailure(message := "Queue must be READY and empty before resetting its former children");
	RETURN;
END_IF

Assert.ThatBool(actual := _Child.Reset(), message := "Counter child must accept cleanup Reset").IsTrue();
END_METHOD

//! <summary>Borrows the concrete class name. Callers must not modify the returned storage.</summary>
{attribute 'monitoring' := 'call'}
PROPERTY ClassName : REFERENCE TO STRING
GET
ClassName REF= _ClassName;
END_GET
END_PROPERTY

//! <summary>Borrows the compiler-initialized namespace name. Callers must not modify it.</summary>
{attribute 'monitoring' := 'call'}
PROPERTY NamespaceName : REFERENCE TO STRING
GET
NamespaceName REF= CurrentNamespace.Name;
END_GET
END_PROPERTY

//! <summary>Reports the complete concrete instance size in bytes.</summary>
{attribute 'monitoring' := 'call'}
PROPERTY SelfSize : ULINT
GET
SelfSize := XSIZEOF(THIS^);
END_GET
END_PROPERTY

END_FUNCTION_BLOCK

// ---- Tests/Tasks/QueueCleanup/TaskQueueCleanupTestGroup.TcPOU
(*
SPDX-FileCopyrightText: © 2026 Oleksandr Tiutyk <trofimich@gmail.com>
SPDX-License-Identifier: MIT
License: https://opensource.org/license/mit
*)

(*!
<summary>Groups the seven independent queue cleanup cases.</summary>
<description>
Owns the cases and their fixed child array for single-task use. Copying invalidates the child bindings.
</description>
*)

{attribute 'no_assign'}
{attribute 'no_explicit_call' := 'do not call this function block directly'}
FUNCTION_BLOCK TaskQueueCleanupTestGroup EXTENDS TOF_Testing.TestGroup<7>
VAR_STAT
	{attribute 'hide'}
	_ClassName : STRING := __POUNAME();
END_VAR
VAR
	_DelayedCleanupAndReuse : TaskQueueCleanupScenarioTest(
		name := "DelayedCleanupAndReuse",
		parent := THIS^,
		scenario := QUEUE_CLEANUP_TEST_SCENARIO.DELAYED_CLEANUP_AND_REUSE
	);
	_RepeatedExecuteFailure : TaskQueueCleanupScenarioTest(
		name := "RepeatedExecuteFailure",
		parent := THIS^,
		scenario := QUEUE_CLEANUP_TEST_SCENARIO.REPEATED_EXECUTE_FAILURE
	);
	_CancelRequestFailure : TaskQueueCleanupScenarioTest(
		name := "CancelRequestFailure",
		parent := THIS^,
		scenario := QUEUE_CLEANUP_TEST_SCENARIO.CANCEL_REQUEST_FAILURE
	);
	_MessageFormattingFailure : TaskQueueCleanupScenarioTest(
		name := "MessageFormattingFailure",
		parent := THIS^,
		scenario := QUEUE_CLEANUP_TEST_SCENARIO.MESSAGE_FORMATTING_FAILURE
	);
	_ExternalCancelDuringCleanup : TaskQueueCleanupScenarioTest(
		name := "ExternalCancelDuringCleanup",
		parent := THIS^,
		scenario := QUEUE_CLEANUP_TEST_SCENARIO.EXTERNAL_CANCEL_DURING_CLEANUP
	);
	_HeldCleanup : TaskQueueCleanupScenarioTest(
		name := "HeldCleanup",
		parent := THIS^,
		scenario := QUEUE_CLEANUP_TEST_SCENARIO.HELD_CLEANUP
	);
	_ExternalCancelWithReleaseFailure : TaskQueueCleanupScenarioTest(
		name := "ExternalCancelWithReleaseFailure",
		parent := THIS^,
		scenario := QUEUE_CLEANUP_TEST_SCENARIO.EXTERNAL_CANCEL_WITH_RELEASE_FAILURE
	);

	_Children : ARRAY [0.._ChildCount - 1] OF TOF_Testing.ITestElement :=
	[
		_DelayedCleanupAndReuse,
		_RepeatedExecuteFailure,
		_CancelRequestFailure,
		_MessageFormattingFailure,
		_ExternalCancelDuringCleanup,
		_HeldCleanup,
		_ExternalCancelWithReleaseFailure
	];
END_VAR

//! <summary>Borrows the fixed child array. Callers must not modify it.</summary>
{attribute 'monitoring' := 'call'}
PROPERTY Children : REFERENCE TO ARRAY [0.._ChildCount - 1] OF TOF_Testing.ITestElement
GET
Children REF= _Children;
END_GET
END_PROPERTY

//! <summary>Borrows the concrete class name. Callers must not modify it.</summary>
{attribute 'monitoring' := 'call'}
PROPERTY ClassName : REFERENCE TO STRING
GET
ClassName REF= _ClassName;
END_GET
END_PROPERTY

//! <summary>Borrows the compiler-initialized namespace name. Callers must not modify it.</summary>
{attribute 'monitoring' := 'call'}
PROPERTY NamespaceName : REFERENCE TO STRING
GET
NamespaceName REF= CurrentNamespace.Name;
END_GET
END_PROPERTY

//! <summary>Reports the complete concrete instance size in bytes.</summary>
{attribute 'monitoring' := 'call'}
PROPERTY SelfSize : ULINT
GET
SelfSize := XSIZEOF(THIS^);
END_GET
END_PROPERTY

END_FUNCTION_BLOCK

// ---- Tests/Tasks/QueueCleanup/TaskQueueCleanupScenarioTest.TcPOU
(*
SPDX-FileCopyrightText: © 2026 Oleksandr Tiutyk <trofimich@gmail.com>
SPDX-License-Identifier: MIT
License: https://opensource.org/license/mit
*)

(*!
<summary>Exercises cooperative queue cleanup under one fault configuration.</summary>
<description>
Owns independent static fixtures. The queue borrows its resource and children and is advanced once per
scenario cycle. The resource is synthetic. AfterTest uses bounded cooperative cancellation before clearing
fixture state. Instances belong to one PLC task and must stay at a stable address.
</description>
*)

{attribute 'no_assign'}
{attribute 'no_explicit_call' := 'do not call this function block directly'}
FUNCTION_BLOCK TaskQueueCleanupScenarioTest EXTENDS TOF_Testing.MultiCycleTest
VAR_STAT
	{attribute 'hide'}
	_ClassName : STRING := __POUNAME();
END_VAR
VAR CONSTANT
	//! <summary>Maximum queue calls per failure or reuse run, including acquisition and release.</summary>
	_MaxRunCycles : UDINT := 32;
	//! <summary>Number of queue calls to observe after the first failure while cleanup is held.</summary>
	_HeldObservationCycles : UINT := 8;
	//! <summary>Allows all remaining synthetic cancellation failures, three child steps and two release steps.</summary>
	_DrainBudget : INT := 16;
END_VAR
VAR
	_Scenario : QUEUE_CLEANUP_TEST_SCENARIO;
	_Phase : QUEUE_CLEANUP_TEST_PHASE;
	_Queue : QueueCleanupQueue(name := "queue");
	_Resource : QueueCleanupResource;
	_Child : QueueCleanupChild;
	_Waiting : CounterTask(name := "waiting");

	_RunStartCycle : UDINT;
	_FirstFailureObserved : BOOL;
	_HeldCycles : UINT;
	_ExpectedExecuteFailures : UINT;
	_ExpectedCancelFailures : UINT;
	_RequestExternalCancel : BOOL;
	_InjectReleaseFailure : BOOL;
	_ExpectedFailureMessage : WSTRING(255);
END_VAR

(*!
<summary>Stores the scenario and selects a cycle budget for both runs.</summary>
<param name="name">Display name of this case.</param>
<param name="parent">Group that owns this test.</param>
<param name="scenario">Independent fault configuration.</param>
*)
METHOD FB_init : BOOL
VAR_INPUT
	bInitRetains: BOOL; // TRUE: the retain variables are initialized (reset warm / reset cold)
	bInCopyCode: BOOL; // TRUE: the instance will be copied to the copy code afterward (online change)
	name : WSTRING;
	parent : TOF_Testing.ITestElement;
	scenario : QUEUE_CLEANUP_TEST_SCENARIO;
END_VAR
_Scenario := scenario;
_Timeout := T#0S;
FB_init := TRUE;
END_METHOD

(*!
<summary>Prepares two borrowed children, configures faults and starts the queue.</summary>
*)
METHOD PROTECTED BeforeTest
_Phase := QUEUE_CLEANUP_TEST_PHASE.FAILURE_RUN;
_RunStartCycle := 0;
_FirstFailureObserved := FALSE;
_HeldCycles := 0;

IF NOT _Queue.State.Ready
	OR_ELSE _Queue.PendingTaskCount <> 0
	OR_ELSE NOT _Child.State.Ready
	OR_ELSE NOT _Waiting.State.Ready
	OR_ELSE _Resource.ResourceAcquired
	OR_ELSE _Resource.ReleaseCalls <> 0
	OR_ELSE _Resource.EarlyRelease
THEN
	RecordFailure(message := "Queue, children and resource must be ready for a new failure run");
	RETURN;
END_IF

_Child.ThrowOnFirstExecute := TRUE;
_Child.ThrowOnGetMessage := _Scenario = QUEUE_CLEANUP_TEST_SCENARIO.MESSAGE_FORMATTING_FAILURE;
_Child.HoldCleanup := _Scenario = QUEUE_CLEANUP_TEST_SCENARIO.HELD_CLEANUP;
_Child.CleanupFailures := 0;
_Child.CancelFailures := 0;
_ExpectedFailureMessage := "First child failure";
_ExpectedExecuteFailures := 1;
_ExpectedCancelFailures := 0;
_InjectReleaseFailure := _Scenario = QUEUE_CLEANUP_TEST_SCENARIO.EXTERNAL_CANCEL_WITH_RELEASE_FAILURE;
_RequestExternalCancel := _InjectReleaseFailure
	OR_ELSE _Scenario = QUEUE_CLEANUP_TEST_SCENARIO.EXTERNAL_CANCEL_DURING_CLEANUP;

